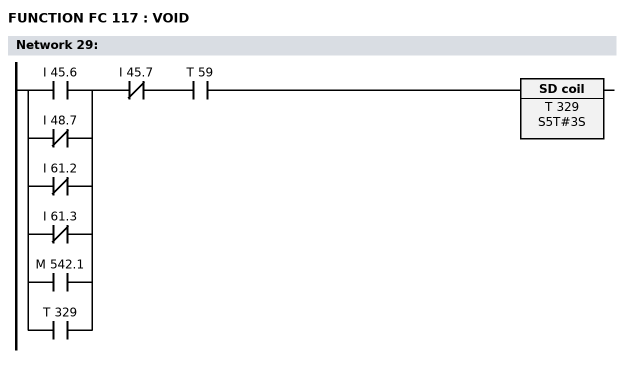

      A(    ;
      O     I     45.6;
      ON    I     48.7;
      ON    I     61.2;
      ON    I     61.3;
      O     M    542.1;
      O     T    329;
      )     ;
      AN    I     45.7;
      A     T     59;
      L     S5T#3S;
      SD    T    329;
NETWORK
TITLE =

      AN    OV;
      =     L      0.0;
      A     L      0.0;
      A     T    329;
      A     M      0.5;
      =     Q     53.6;
      A     L      0.0;
      AN    T    329;
      A(    ;
      O     T    309;
      O     T     69;
      )     ;
      =     Q     53.7;
      A     L      0.0;
      A     I     48.7;
      A     I     61.2;
      A     I     61.3;
      =     L      0.1;
      A     L      0.1;
      A     DB49.DBX    9.2;
      AN    DB49.DBX    9.3;
      =     L      0.2;
      A     L      0.2;
      BLD   102;
      L     S5T#3S;
      SD    T    309;
      A     L      0.2;
      A     T    309;
      =     DB49.DBX    9.4;
      A     L      0.1;
      A     DB49.DBX    9.3;
      AN    DB49.DBX    9.2;
      =     L      0.2;
      A     L      0.2;
      BLD   102;
      L     S5T#3S;
      SD    T     69;
      A     L      0.2;
      A     T     69;
      =     DB49.DBX    9.5;
NETWORK
TITLE =
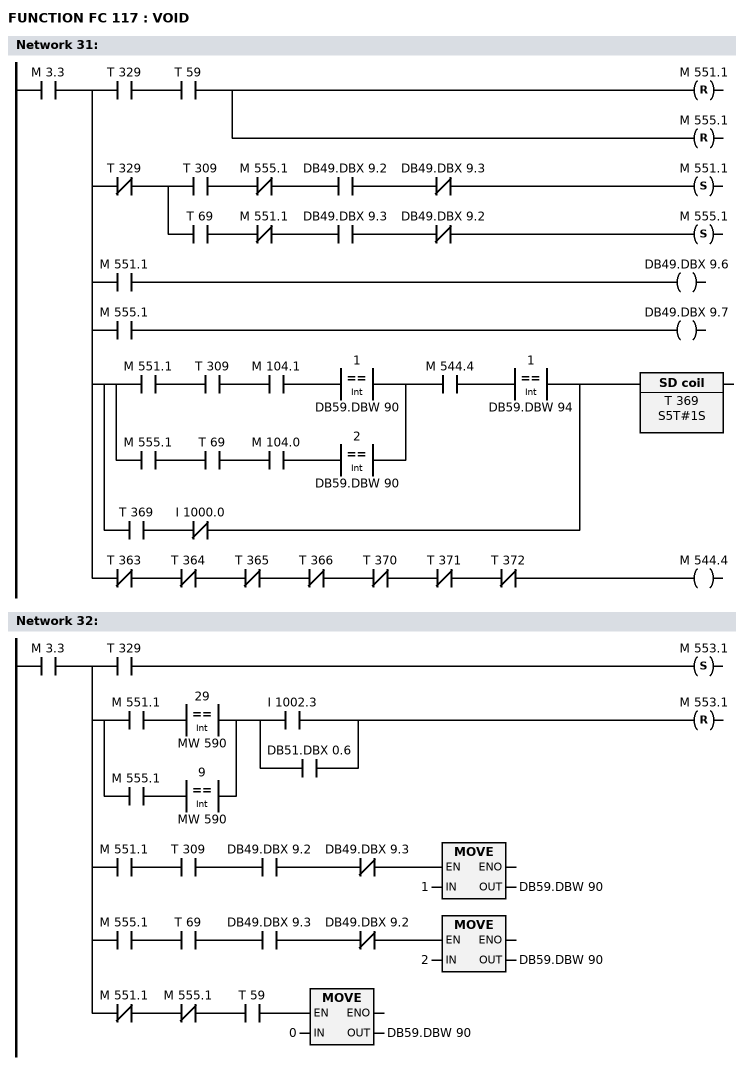

      A     M      3.3;
      =     L      0.0;
      A     L      0.0;
      A     T    329;
      A     T     59;
      R     M    551.1;
      R     M    555.1;
      A     L      0.0;
      AN    T    329;
      =     L      0.1;
      A     L      0.1;
      A     T    309;
      AN    M    555.1;
      A     DB49.DBX    9.2;
      AN    DB49.DBX    9.3;
      S     M    551.1;
      A     L      0.1;
      A     T     69;
      AN    M    551.1;
      A     DB49.DBX    9.3;
      AN    DB49.DBX    9.2;
      S     M    555.1;
      A     L      0.0;
      A     M    551.1;
      =     DB49.DBX    9.6;
      A     L      0.0;
      A     M    555.1;
      =     DB49.DBX    9.7;
      A     L      0.0;
      A(    ;
      A(    ;
      A     M    551.1;
      A     T    309;
      A     M    104.1;
      A(    ;
      L     1;
      L     DB59.DBW   90;
      ==I   ;
      )     ;
      O     ;
      A     M    555.1;
      A     T     69;
      A     M    104.0;
      A(    ;
      L     2;
      L     DB59.DBW   90;
      ==I   ;
      )     ;
      )     ;
      A     M    544.4;
      A(    ;
      L     1;
      L     DB59.DBW   94;
      ==I   ;
      )     ;
      O     ;
      A     T    369;
      AN    I   1000.0;
      )     ;
      L     S5T#1S;
      SD    T    369;
      A     L      0.0;
      AN    T    363;
      AN    T    364;
      AN    T    365;
      AN    T    366;
      AN    T    370;
      AN    T    371;
      AN    T    372;
      =     M    544.4;
NETWORK
TITLE =

      A     M      3.3;
      =     L      0.0;
      A     L      0.0;
      A     T    329;
      S     M    553.1;
      A     L      0.0;
      A(    ;
      A     M    551.1;
      A(    ;
      L     29;
      L     MW   590;
      ==I   ;
      )     ;
      O     ;
      A     M    555.1;
      A(    ;
      L     9;
      L     MW   590;
      ==I   ;
      )     ;
      )     ;
      A(    ;
      O     I   1002.3;
      O     DB51.DBX    0.6;
      )     ;
      R     M    553.1;
      A     L      0.0;
      A     M    551.1;
      A     T    309;
      A     DB49.DBX    9.2;
      AN    DB49.DBX    9.3;
      JNB   _00d;
      L     1;
      T     DB59.DBW   90;
_00d: NOP   0;
      A     L      0.0;
      A     M    555.1;
      A     T     69;
      A     DB49.DBX    9.3;
      AN    DB49.DBX    9.2;
      JNB   _00e;
      L     2;
      T     DB59.DBW   90;
_00e: NOP   0;
      A     L      0.0;
      AN    M    551.1;
      AN    M    555.1;
      A     T     59;
      JNB   _00f;
      L     0;
      T     DB59.DBW   90;
_00f: NOP   0;
NETWORK
TITLE =

      AN    OV;
      =     L      0.0;
      A     L      0.0;
      A(    ;
      A     T    330;
      A     DB49.DBX    2.1;
      A     DB49.DBX   10.0;
      O     ;
      A     M    580.0;
      A     M    580.1;
      O     ;
      AN    M    580.0;
      AN    M    580.1;
      )     ;
      S     M    580.0;
      R     M    580.1;
      A     L      0.0;
      A     T    330;
      A     DB49.DBX    2.1;
      A     DB49.DBX   10.1;
      S     M    580.1;
      R     M    580.0;
      A     L      0.0;
      A     M    580.0;
      =     DB49.DBX   10.2;
      A     L      0.0;
      A     M    580.1;
      =     DB49.DBX   10.3;
NETWORK
TITLE =

      AN    OV;
      =     L      0.0;
      A     L      0.0;
      A(    ;
      A     I     62.0;
      AN    I     62.1;
      O     ;
      AN    I     62.0;
      A     I     62.1;
      O     ;
      AN    I     62.0;
      AN    I     62.1;
      A     I     49.3;
      )     ;
      =     L      0.1;
      A     L      0.1;
      A     T    350;
      =     DB49.DBX    0.5;
      A     L      0.1;
      BLD   102;
      L     S5T#2S;
      SD    T    350;
      A     L      0.0;
      A(    ;
      A     DB49.DBX   10.2;
      A     I     61.1;
      O     ;
      A     DB49.DBX   10.3;
      AN    I     61.1;
      )     ;
      A     I     62.0;
      A     I     62.1;
      A     I     49.3;
      AN    T    330;
      =     L      0.1;
      A     L      0.1;
      A     T    420;
      =     DB49.DBX    1.5;
      A     L      0.1;
      BLD   102;
      L     S5T#3S;
      SD    T    420;
NETWORK
TITLE =
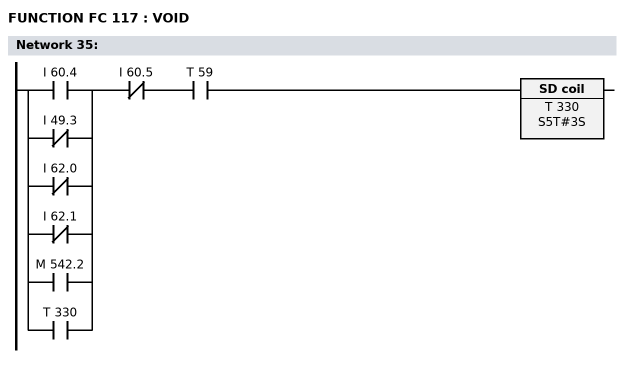

      A(    ;
      O     I     60.4;
      ON    I     49.3;
      ON    I     62.0;
      ON    I     62.1;
      O     M    542.2;
      O     T    330;
      )     ;
      AN    I     60.5;
      A     T     59;
      L     S5T#3S;
      SD    T    330;
NETWORK
TITLE =

      AN    OV;
      =     L      0.0;
      A     L      0.0;
      A     T    330;
      A     M      0.5;
      =     Q     56.4;
      A     L      0.0;
      AN    T    330;
      A(    ;
      O     T    310;
      O     T     70;
      )     ;
      =     Q     56.5;
      A     L      0.0;
      A     I     49.3;
      A     I     62.0;
      A     I     62.1;
      =     L      0.1;
      A     L      0.1;
      A     DB49.DBX   10.2;
      AN    DB49.DBX   10.3;
      =     L      0.2;
      A     L      0.2;
      BLD   102;
      L     S5T#3S;
      SD    T    310;
      A     L      0.2;
      A     T    310;
      =     DB49.DBX   10.4;
      A     L      0.1;
      A     DB49.DBX   10.3;
      AN    DB49.DBX   10.2;
      =     L      0.2;
      A     L      0.2;
      BLD   102;
      L     S5T#3S;
      SD    T     70;
      A     L      0.2;
      A     T     70;
      =     DB49.DBX   10.5;
NETWORK
TITLE =
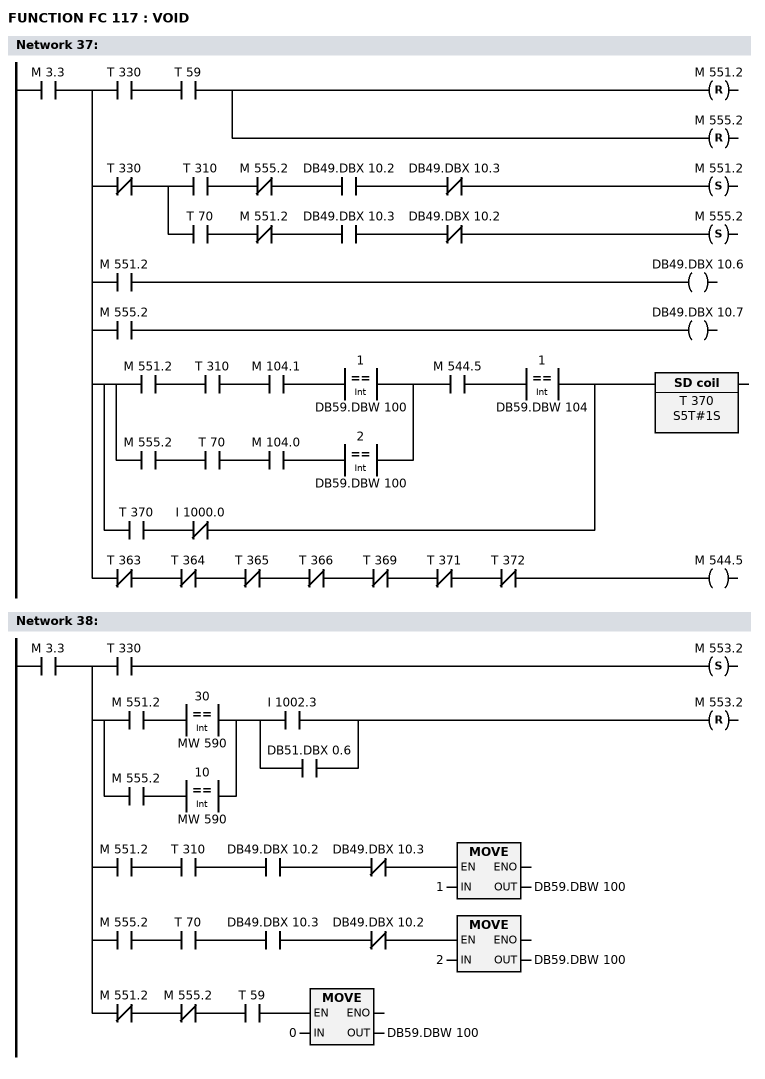

      A     M      3.3;
      =     L      0.0;
      A     L      0.0;
      A     T    330;
      A     T     59;
      R     M    551.2;
      R     M    555.2;
      A     L      0.0;
      AN    T    330;
      =     L      0.1;
      A     L      0.1;
      A     T    310;
      AN    M    555.2;
      A     DB49.DBX   10.2;
      AN    DB49.DBX   10.3;
      S     M    551.2;
      A     L      0.1;
      A     T     70;
      AN    M    551.2;
      A     DB49.DBX   10.3;
      AN    DB49.DBX   10.2;
      S     M    555.2;
      A     L      0.0;
      A     M    551.2;
      =     DB49.DBX   10.6;
      A     L      0.0;
      A     M    555.2;
      =     DB49.DBX   10.7;
      A     L      0.0;
      A(    ;
      A(    ;
      A     M    551.2;
      A     T    310;
      A     M    104.1;
      A(    ;
      L     1;
      L     DB59.DBW  100;
      ==I   ;
      )     ;
      O     ;
      A     M    555.2;
      A     T     70;
      A     M    104.0;
      A(    ;
      L     2;
      L     DB59.DBW  100;
      ==I   ;
      )     ;
      )     ;
      A     M    544.5;
      A(    ;
      L     1;
      L     DB59.DBW  104;
      ==I   ;
      )     ;
      O     ;
      A     T    370;
      AN    I   1000.0;
      )     ;
      L     S5T#1S;
      SD    T    370;
      A     L      0.0;
      AN    T    363;
      AN    T    364;
      AN    T    365;
      AN    T    366;
      AN    T    369;
      AN    T    371;
      AN    T    372;
      =     M    544.5;
NETWORK
TITLE =

      A     M      3.3;
      =     L      0.0;
      A     L      0.0;
      A     T    330;
      S     M    553.2;
      A     L      0.0;
      A(    ;
      A     M    551.2;
      A(    ;
      L     30;
      L     MW   590;
      ==I   ;
      )     ;
      O     ;
      A     M    555.2;
      A(    ;
      L     10;
      L     MW   590;
      ==I   ;
      )     ;
      )     ;
      A(    ;
      O     I   1002.3;
      O     DB51.DBX    0.6;
      )     ;
      R     M    553.2;
      A     L      0.0;
      A     M    551.2;
      A     T    310;
      A     DB49.DBX   10.2;
      AN    DB49.DBX   10.3;
      JNB   _010;
      L     1;
      T     DB59.DBW  100;
_010: NOP   0;
      A     L      0.0;
      A     M    555.2;
      A     T     70;
      A     DB49.DBX   10.3;
      AN    DB49.DBX   10.2;
      JNB   _011;
      L     2;
      T     DB59.DBW  100;
_011: NOP   0;
      A     L      0.0;
      AN    M    551.2;
      AN    M    555.2;
      A     T     59;
      JNB   _012;
      L     0;
      T     DB59.DBW  100;
_012: NOP   0;
NETWORK
TITLE =

      AN    OV;
      =     L      0.0;
      A     L      0.0;
      A(    ;
      A     T    331;
      A     DB49.DBX    2.1;
      A     DB49.DBX   11.0;
      O     ;
      A     M    581.0;
      A     M    581.1;
      O     ;
      AN    M    581.0;
      AN    M    581.1;
      )     ;
      S     M    581.0;
      R     M    581.1;
      A     L      0.0;
      A     T    331;
      A     DB49.DBX    2.1;
      A     DB49.DBX   11.1;
      S     M    581.1;
      R     M    581.0;
      A     L      0.0;
      A     M    581.0;
      =     DB49.DBX   11.2;
      A     L      0.0;
      A     M    581.1;
      =     DB49.DBX   11.3;
NETWORK
TITLE =

      AN    OV;
      =     L      0.0;
      A     L      0.0;
      A(    ;
      A     I     61.4;
      AN    I     61.5;
      O     ;
      AN    I     61.4;
      A     I     61.5;
      O     ;
      AN    I     61.4;
      AN    I     61.5;
      A     I     49.0;
      )     ;
      =     L      0.1;
      A     L      0.1;
      A     T    351;
      =     DB49.DBX    0.6;
      A     L      0.1;
      BLD   102;
      L     S5T#2S;
      SD    T    351;
      A     L      0.0;
      A(    ;
      A     DB49.DBX   11.2;
      A     I     61.6;
      O     ;
      A     DB49.DBX   11.3;
      AN    I     61.6;
      )     ;
      A     I     61.4;
      A     I     61.5;
      A     I     49.0;
      AN    T    331;
      =     L      0.1;
      A     L      0.1;
      A     T    421;
      =     DB49.DBX    1.6;
      A     L      0.1;
      BLD   102;
      L     S5T#3S;
      SD    T    421;
NETWORK
TITLE =
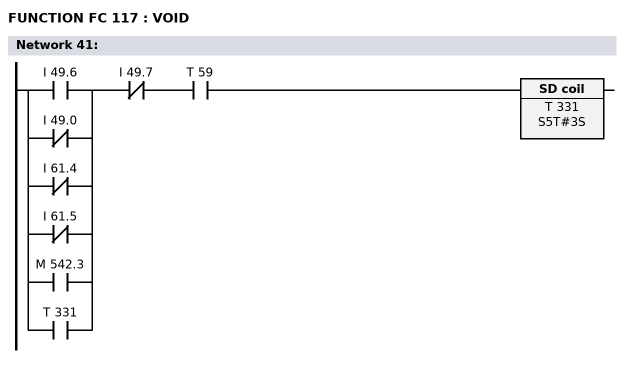

      A(    ;
      O     I     49.6;
      ON    I     49.0;
      ON    I     61.4;
      ON    I     61.5;
      O     M    542.3;
      O     T    331;
      )     ;
      AN    I     49.7;
      A     T     59;
      L     S5T#3S;
      SD    T    331;
NETWORK
TITLE =

      AN    OV;
      =     L      0.0;
      A     L      0.0;
      A     T    331;
      A     M      0.5;
      =     Q     56.0;
      A     L      0.0;
      AN    T    331;
      A(    ;
      O     T    311;
      O     T     71;
      )     ;
      =     Q     56.1;
      A     L      0.0;
      A     I     49.0;
      A     I     61.4;
      A     I     61.5;
      =     L      0.1;
      A     L      0.1;
      A     DB49.DBX   11.2;
      AN    DB49.DBX   11.3;
      =     L      0.2;
      A     L      0.2;
      BLD   102;
      L     S5T#3S;
      SD    T    311;
      A     L      0.2;
      A     T    311;
      =     DB49.DBX   11.4;
      A     L      0.1;
      A     DB49.DBX   11.3;
      AN    DB49.DBX   11.2;
      =     L      0.2;
      A     L      0.2;
      BLD   102;
      L     S5T#3S;
      SD    T     71;
      A     L      0.2;
      A     T     71;
      =     DB49.DBX   11.5;
NETWORK
TITLE =
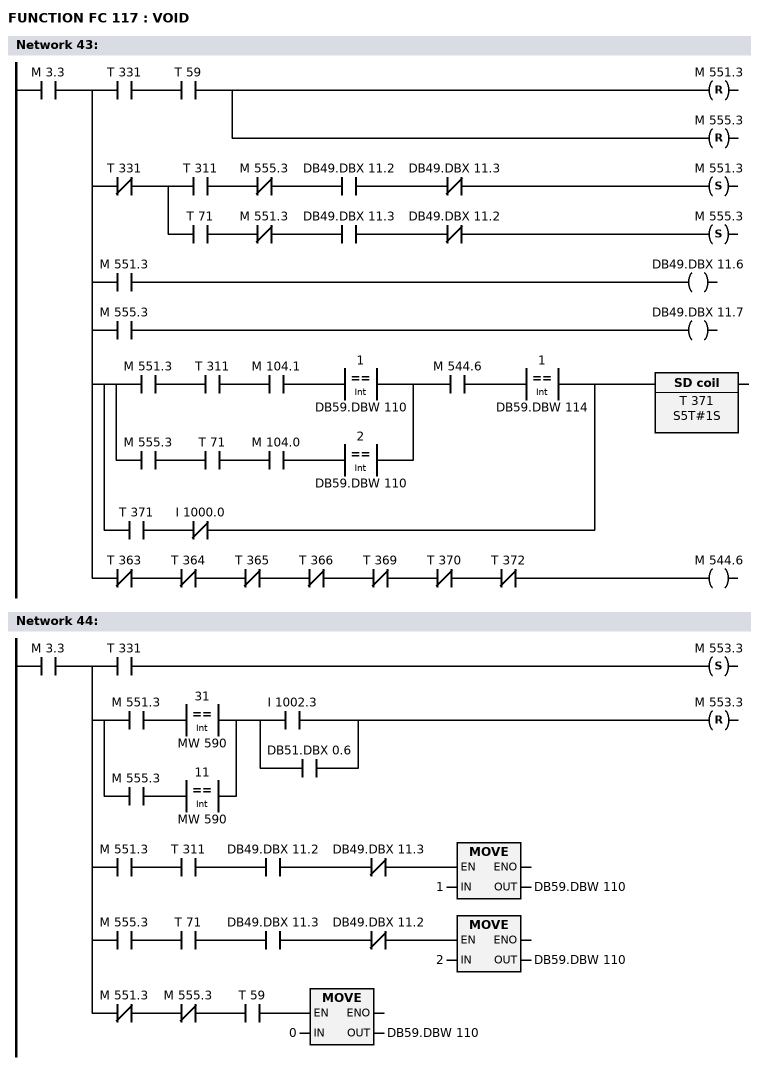

      A     M      3.3;
      =     L      0.0;
      A     L      0.0;
      A     T    331;
      A     T     59;
      R     M    551.3;
      R     M    555.3;
      A     L      0.0;
      AN    T    331;
      =     L      0.1;
      A     L      0.1;
      A     T    311;
      AN    M    555.3;
      A     DB49.DBX   11.2;
      AN    DB49.DBX   11.3;
      S     M    551.3;
      A     L      0.1;
      A     T     71;
      AN    M    551.3;
      A     DB49.DBX   11.3;
      AN    DB49.DBX   11.2;
      S     M    555.3;
      A     L      0.0;
      A     M    551.3;
      =     DB49.DBX   11.6;
      A     L      0.0;
      A     M    555.3;
      =     DB49.DBX   11.7;
      A     L      0.0;
      A(    ;
      A(    ;
      A     M    551.3;
      A     T    311;
      A     M    104.1;
      A(    ;
      L     1;
      L     DB59.DBW  110;
      ==I   ;
      )     ;
      O     ;
      A     M    555.3;
      A     T     71;
      A     M    104.0;
      A(    ;
      L     2;
      L     DB59.DBW  110;
      ==I   ;
      )     ;
      )     ;
      A     M    544.6;
      A(    ;
      L     1;
      L     DB59.DBW  114;
      ==I   ;
      )     ;
      O     ;
      A     T    371;
      AN    I   1000.0;
      )     ;
      L     S5T#1S;
      SD    T    371;
      A     L      0.0;
      AN    T    363;
      AN    T    364;
      AN    T    365;
      AN    T    366;
      AN    T    369;
      AN    T    370;
      AN    T    372;
      =     M    544.6;
NETWORK
TITLE =

      A     M      3.3;
      =     L      0.0;
      A     L      0.0;
      A     T    331;
      S     M    553.3;
      A     L      0.0;
      A(    ;
      A     M    551.3;
      A(    ;
      L     31;
      L     MW   590;
      ==I   ;
      )     ;
      O     ;
      A     M    555.3;
      A(    ;
      L     11;
      L     MW   590;
      ==I   ;
      )     ;
      )     ;
      A(    ;
      O     I   1002.3;
      O     DB51.DBX    0.6;
      )     ;
      R     M    553.3;
      A     L      0.0;
      A     M    551.3;
      A     T    311;
      A     DB49.DBX   11.2;
      AN    DB49.DBX   11.3;
      JNB   _013;
      L     1;
      T     DB59.DBW  110;
_013: NOP   0;
      A     L      0.0;
      A     M    555.3;
      A     T     71;
      A     DB49.DBX   11.3;
      AN    DB49.DBX   11.2;
      JNB   _014;
      L     2;
      T     DB59.DBW  110;
_014: NOP   0;
      A     L      0.0;
      AN    M    551.3;
      AN    M    555.3;
      A     T     59;
      JNB   _015;
      L     0;
      T     DB59.DBW  110;
_015: NOP   0;
NETWORK
TITLE =

      AN    OV;
      =     L      0.0;
      A     L      0.0;
      A(    ;
      A     T    332;
      A     DB49.DBX    2.1;
      A     DB49.DBX   12.0;
      O     ;
      A     M    582.0;
      A     M    582.1;
      O     ;
      AN    M    582.0;
      AN    M    582.1;
      )     ;
      S     M    582.0;
      R     M    582.1;
      A     L      0.0;
      A     T    332;
      A     DB49.DBX    2.1;
      A     DB49.DBX   12.1;
      S     M    582.1;
      R     M    582.0;
      A     L      0.0;
      A     M    582.0;
      =     DB49.DBX   12.2;
      A     L      0.0;
      A     M    582.1;
      =     DB49.DBX   12.3;
NETWORK
TITLE =

      AN    OV;
      =     L      0.0;
      A     L      0.0;
      A(    ;
      A     I     62.2;
      AN    I     62.3;
      O     ;
      AN    I     62.2;
      A     I     62.3;
      O     ;
      AN    I     62.2;
      AN    I     62.3;
      A     I     49.4;
      )     ;
      =     L      0.1;
      A     L      0.1;
      A     T    352;
      =     DB49.DBX    0.7;
      A     L      0.1;
      BLD   102;
      L     S5T#2S;
      SD    T    352;
      A     L      0.0;
      A(    ;
      A     DB49.DBX   12.2;
      A     I     61.7;
      O     ;
      A     DB49.DBX   12.3;
      AN    I     61.7;
      )     ;
      A     I     62.2;
      A     I     62.3;
      A     I     49.4;
      AN    T    332;
      =     L      0.1;
      A     L      0.1;
      A     T    422;
      =     DB49.DBX    1.7;
      A     L      0.1;
      BLD   102;
      L     S5T#3S;
      SD    T    422;
NETWORK
TITLE =
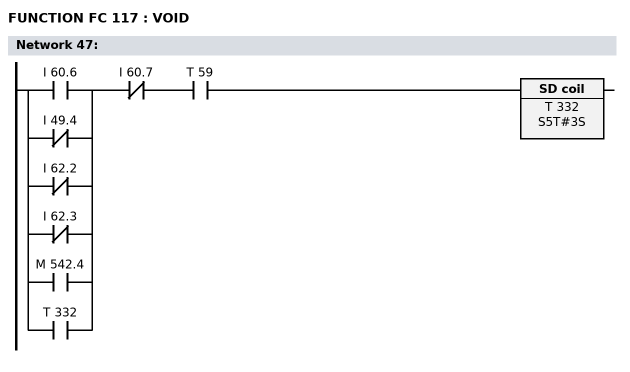

      A(    ;
      O     I     60.6;
      ON    I     49.4;
      ON    I     62.2;
      ON    I     62.3;
      O     M    542.4;
      O     T    332;
      )     ;
      AN    I     60.7;
      A     T     59;
      L     S5T#3S;
      SD    T    332;
NETWORK
TITLE =

      AN    OV;
      =     L      0.0;
      A     L      0.0;
      A     T    332;
      A     M      0.5;
      =     Q     56.6;
      A     L      0.0;
      AN    T    332;
      A(    ;
      O     T    312;
      O     T     72;
      )     ;
      =     Q     56.7;
      A     L      0.0;
      A     I     49.4;
      A     I     62.2;
      A     I     62.3;
      =     L      0.1;
      A     L      0.1;
      A     DB49.DBX   12.2;
      AN    DB49.DBX   12.3;
      =     L      0.2;
      A     L      0.2;
      BLD   102;
      L     S5T#3S;
      SD    T    312;
      A     L      0.2;
      A     T    312;
      =     DB49.DBX   12.4;
      A     L      0.1;
      A     DB49.DBX   12.3;
      AN    DB49.DBX   12.2;
      =     L      0.2;
      A     L      0.2;
      BLD   102;
      L     S5T#3S;
      SD    T     72;
      A     L      0.2;
      A     T     72;
      =     DB49.DBX   12.5;
NETWORK
TITLE =
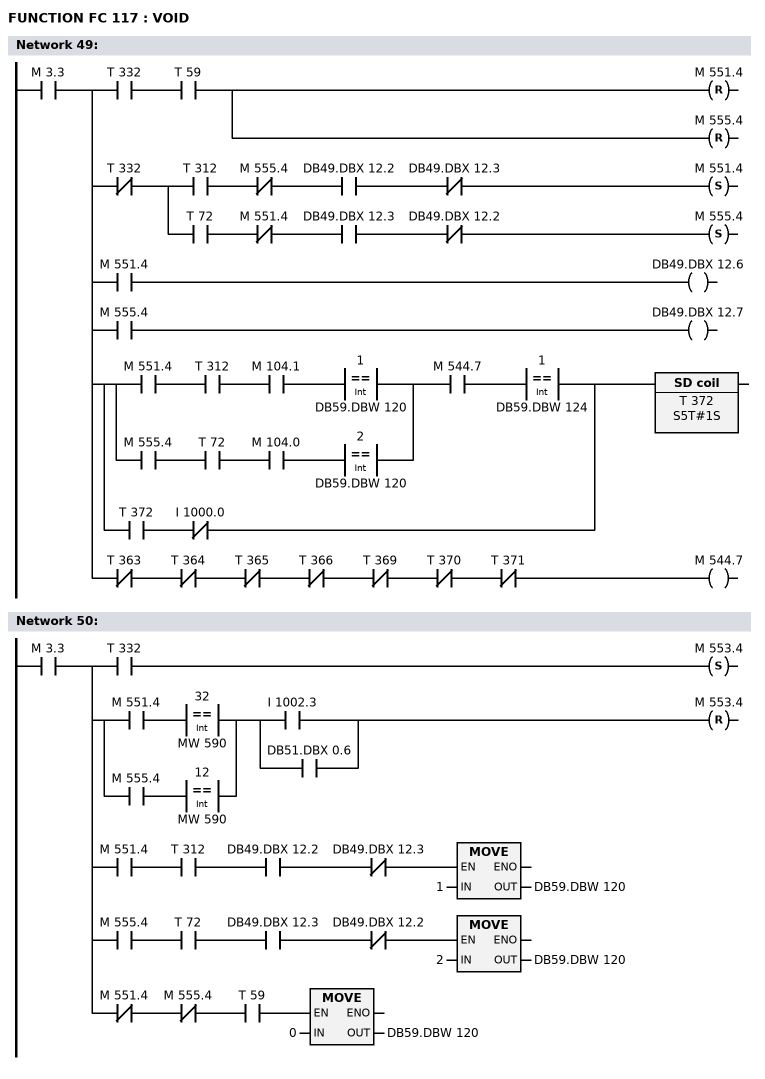

      A     M      3.3;
      =     L      0.0;
      A     L      0.0;
      A     T    332;
      A     T     59;
      R     M    551.4;
      R     M    555.4;
      A     L      0.0;
      AN    T    332;
      =     L      0.1;
      A     L      0.1;
      A     T    312;
      AN    M    555.4;
      A     DB49.DBX   12.2;
      AN    DB49.DBX   12.3;
      S     M    551.4;
      A     L      0.1;
      A     T     72;
      AN    M    551.4;
      A     DB49.DBX   12.3;
      AN    DB49.DBX   12.2;
      S     M    555.4;
      A     L      0.0;
      A     M    551.4;
      =     DB49.DBX   12.6;
      A     L      0.0;
      A     M    555.4;
      =     DB49.DBX   12.7;
      A     L      0.0;
      A(    ;
      A(    ;
      A     M    551.4;
      A     T    312;
      A     M    104.1;
      A(    ;
      L     1;
      L     DB59.DBW  120;
      ==I   ;
      )     ;
      O     ;
      A     M    555.4;
      A     T     72;
      A     M    104.0;
      A(    ;
      L     2;
      L     DB59.DBW  120;
      ==I   ;
      )     ;
      )     ;
      A     M    544.7;
      A(    ;
      L     1;
      L     DB59.DBW  124;
      ==I   ;
      )     ;
      O     ;
      A     T    372;
      AN    I   1000.0;
      )     ;
      L     S5T#1S;
      SD    T    372;
      A     L      0.0;
      AN    T    363;
      AN    T    364;
      AN    T    365;
      AN    T    366;
      AN    T    369;
      AN    T    370;
      AN    T    371;
      =     M    544.7;
NETWORK
TITLE =

      A     M      3.3;
      =     L      0.0;
      A     L      0.0;
      A     T    332;
      S     M    553.4;
      A     L      0.0;
      A(    ;
      A     M    551.4;
      A(    ;
      L     32;
      L     MW   590;
      ==I   ;
      )     ;
      O     ;
      A     M    555.4;
      A(    ;
      L     12;
      L     MW   590;
      ==I   ;
      )     ;
      )     ;
      A(    ;
      O     I   1002.3;
      O     DB51.DBX    0.6;
      )     ;
      R     M    553.4;
      A     L      0.0;
      A     M    551.4;
      A     T    312;
      A     DB49.DBX   12.2;
      AN    DB49.DBX   12.3;
      JNB   _016;
      L     1;
      T     DB59.DBW  120;
_016: NOP   0;
      A     L      0.0;
      A     M    555.4;
      A     T     72;
      A     DB49.DBX   12.3;
      AN    DB49.DBX   12.2;
      JNB   _017;
      L     2;
      T     DB59.DBW  120;
_017: NOP   0;
      A     L      0.0;
      AN    M    551.4;
      AN    M    555.4;
      A     T     59;
      JNB   _018;
      L     0;
      T     DB59.DBW  120;
_018: NOP   0;
NETWORK
TITLE =

      AN    OV;
      =     L      0.0;
      A     L      0.0;
      A     I     45.1;
      L     S5T#3S;
      SD    T    158;
      A     L      0.0;
      A     I     44.3;
      L     S5T#3S;
      SD    T    159;
      A     L      0.0;
      A     I     45.3;
      L     S5T#3S;
      SD    T    160;
      A     L      0.0;
      A     I     44.5;
      L     S5T#3S;
      SD    T    161;
      A     L      0.0;
      A     I     45.7;
      L     S5T#3S;
      SD    T    164;
      A     L      0.0;
      A     I     60.5;
      L     S5T#3S;
      SD    T    165;
      A     L      0.0;
      A     I     49.7;
      L     S5T#3S;
      SD    T    166;
      A     L      0.0;
      A     I     60.7;
      L     S5T#3S;
      SD    T    167;
NETWORK
TITLE =

      AN    OV;
      =     L      0.0;
      A     L      0.0;
      A(    ;
      O(    ;
      L     23;
      L     MW   590;
      ==I   ;
      )     ;
      O(    ;
      L     3;
      L     MW   590;
      ==I   ;
      )     ;
      )     ;
      A     I   1003.6;
      =     M    541.3;
      A     L      0.0;
      A(    ;
      O(    ;
      L     24;
      L     MW   590;
      ==I   ;
      )     ;
      O(    ;
      L     4;
      L     MW   590;
      ==I   ;
      )     ;
      )     ;
      A     I   1003.6;
      =     M    541.4;
      A     L      0.0;
      A(    ;
      O(    ;
      L     25;
      L     MW   590;
      ==I   ;
      )     ;
      O(    ;
      L     5;
      L     MW   590;
      ==I   ;
      )     ;
      )     ;
      A     I   1003.6;
      =     M    541.5;
      A     L      0.0;
      A(    ;
      O(    ;
      L     26;
      L     MW   590;
      ==I   ;
      )     ;
      O(    ;
      L     6;
      L     MW   590;
      ==I   ;
      )     ;
      )     ;
      A     I   1003.6;
      =     M    541.6;
      A     L      0.0;
      A(    ;
      O(    ;
      L     29;
      L     MW   590;
      ==I   ;
      )     ;
      O(    ;
      L     9;
      L     MW   590;
      ==I   ;
      )     ;
      )     ;
      A     I   1003.6;
      =     M    542.1;
      A     L      0.0;
      A(    ;
      O(    ;
      L     30;
      L     MW   590;
      ==I   ;
      )     ;
      O(    ;
      L     10;
      L     MW   590;
      ==I   ;
      )     ;
      )     ;
      A     I   1003.6;
      =     M    542.2;
      A     L      0.0;
      A(    ;
      O(    ;
      L     31;
      L     MW   590;
      ==I   ;
      )     ;
      O(    ;
      L     11;
      L     MW   590;
      ==I   ;
      )     ;
      )     ;
      A     I   1003.6;
      =     M    542.3;
      A     L      0.0;
      A(    ;
      O(    ;
      L     32;
      L     MW   590;
      ==I   ;
      )     ;
      O(    ;
      L     12;
      L     MW   590;
      ==I   ;
      )     ;
      )     ;
      A     I   1003.6;
      =     M    542.4;
NETWORK
TITLE =

      A     M      3.3;
      =     L      0.0;
      BLD   103;
      CALL FB   515 , DB   200 (
           STN_V_ACTIVE             := L      0.0,
           PLT_Amount               := 12,
           PLT1_Code                := 0,
           PLT2_Code                := 0,
           PLT3_Code                := DB59.DBW   30,
           PLT4_Code                := DB59.DBW   40,
           PLT5_Code                := DB59.DBW   50,
           PLT6_Code                := DB59.DBW   60,
           PLT9_Code                := DB59.DBW   90,
           PLT10_Code               := DB59.DBW  100,
           PLT11_Code               := DB59.DBW  110,
           PLT12_Code               := DB59.DBW  120,
           PLT13_Code               := 0,
           PLT14_Code               := 0,
           PLT15_Code               := 0,
           PLT16_Code               := 0,
           PLT17_Code               := 0,
           PLT18_Code               := 0,
           PLT19_Code               := 0,
           PLT20_Code               := 0,
           PLT3_Priority            := DB59.DBW   34,
           PLT4_Priority            := DB59.DBW   44,
           PLT5_Priority            := DB59.DBW   54,
           PLT6_Priority            := DB59.DBW   64,
           PLT9_Priority            := DB59.DBW   94,
           PLT10_Priority           := DB59.DBW  104,
           PLT11_Priority           := DB59.DBW  114,
           PLT12_Priority           := DB59.DBW  124);

      NOP   0;
END_FUNCTION

FUNCTION FC 118 : VOID
TITLE =
VERSION : 0.1

BEGIN
NETWORK
TITLE =
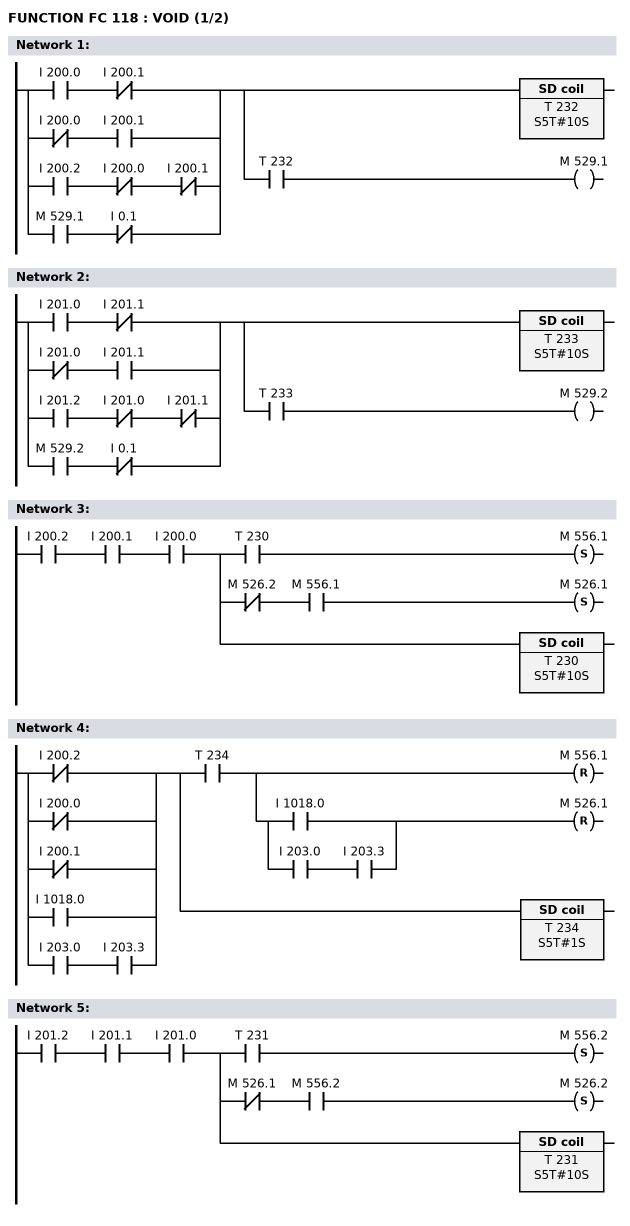

      A     I    200.0;
      AN    I    200.1;
      O     ;
      AN    I    200.0;
      A     I    200.1;
      O     ;
      A     I    200.2;
      AN    I    200.0;
      AN    I    200.1;
      O     ;
      A     M    529.1;
      AN    I      0.1;
      =     L      0.0;
      A     L      0.0;
      BLD   102;
      L     S5T#10S;
      SD    T    232;
      A     L      0.0;
      A     T    232;
      =     M    529.1;
NETWORK
TITLE =

      A     I    201.0;
      AN    I    201.1;
      O     ;
      AN    I    201.0;
      A     I    201.1;
      O     ;
      A     I    201.2;
      AN    I    201.0;
      AN    I    201.1;
      O     ;
      A     M    529.2;
      AN    I      0.1;
      =     L      0.0;
      A     L      0.0;
      BLD   102;
      L     S5T#10S;
      SD    T    233;
      A     L      0.0;
      A     T    233;
      =     M    529.2;
NETWORK
TITLE =

      A     I    200.2;
      A     I    200.1;
      A     I    200.0;
      =     L      0.0;
      A     L      0.0;
      A     T    230;
      S     M    556.1;
      A     L      0.0;
      AN    M    526.2;
      A     M    556.1;
      S     M    526.1;
      A     L      0.0;
      BLD   102;
      L     S5T#10S;
      SD    T    230;
NETWORK
TITLE =

      ON    I    200.2;
      ON    I    200.0;
      ON    I    200.1;
      O     I   1018.0;
      O     ;
      A     I    203.0;
      A     I    203.3;
      =     L      0.0;
      A     L      0.0;
      A     T    234;
      =     L      0.1;
      A     L      0.1;
      BLD   102;
      R     M    556.1;
      A     L      0.1;
      A(    ;
      O     I   1018.0;
      O     ;
      A     I    203.0;
      A     I    203.3;
      )     ;
      R     M    526.1;
      A     L      0.0;
      BLD   102;
      L     S5T#1S;
      SD    T    234;
NETWORK
TITLE =

      A     I    201.2;
      A     I    201.1;
      A     I    201.0;
      =     L      0.0;
      A     L      0.0;
      A     T    231;
      S     M    556.2;
      A     L      0.0;
      AN    M    526.1;
      A     M    556.2;
      S     M    526.2;
      A     L      0.0;
      BLD   102;
      L     S5T#10S;
      SD    T    231;
NETWORK
TITLE =
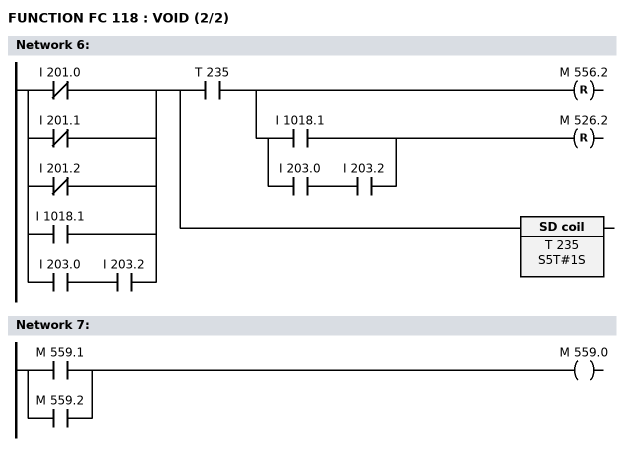

      ON    I    201.0;
      ON    I    201.1;
      ON    I    201.2;
      O     I   1018.1;
      O     ;
      A     I    203.0;
      A     I    203.2;
      =     L      0.0;
      A     L      0.0;
      A     T    235;
      =     L      0.1;
      A     L      0.1;
      BLD   102;
      R     M    556.2;
      A     L      0.1;
      A(    ;
      O     I   1018.1;
      O     ;
      A     I    203.0;
      A     I    203.2;
      )     ;
      R     M    526.2;
      A     L      0.0;
      BLD   102;
      L     S5T#1S;
      SD    T    235;
NETWORK
TITLE =

      O     M    559.1;
      O     M    559.2;
      =     M    559.0;
NETWORK
TITLE =

      AN    OV;
      =     L      0.0;
      A     L      0.0;
      A     M    559.4;
      AN    M    556.1;
      S     M    559.1;
      A     L      0.0;
      A(    ;
      A     M    556.1;
      A     T    230;
      O     ;
      A     I    203.0;
      A     I    203.3;
      O     ;
      AN    I    201.2;
      AN    I    200.0;
      AN    I    200.1;
      O     ;
      AN    I    201.1;
      AN    I    201.0;
      AN    I    200.2;
      )     ;
      R     M    559.1;
NETWORK
TITLE =

      AN    OV;
      =     L      0.0;
      A     L      0.0;
      A     M    559.3;
      AN    M    556.2;
      S     M    559.2;
      A     L      0.0;
      A(    ;
      A     M    556.2;
      A     T    231;
      O     ;
      A     I    203.0;
      A     I    203.2;
      O     ;
      AN    I    200.2;
      AN    I    201.1;
      AN    I    201.0;
      O     ;
      AN    I    200.0;
      AN    I    200.1;
      AN    I    201.2;
      )     ;
      R     M    559.2;
NETWORK
TITLE =
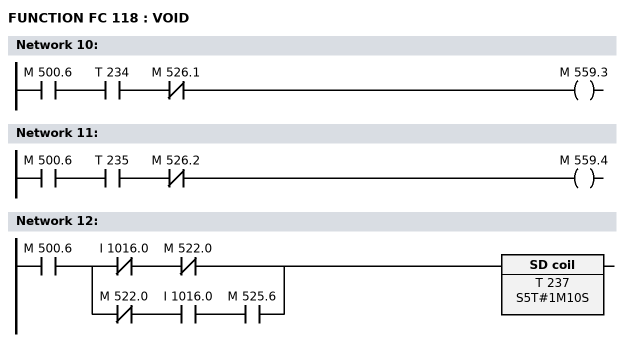

      A     M    500.6;
      A     T    234;
      AN    M    526.1;
      =     M    559.3;
NETWORK
TITLE =

      A     M    500.6;
      A     T    235;
      AN    M    526.2;
      =     M    559.4;
NETWORK
TITLE =

      A     M    500.6;
      A(    ;
      AN    I   1016.0;
      AN    M    522.0;
      O     ;
      AN    M    522.0;
      A     I   1016.0;
      A     M    525.6;
      )     ;
      L     S5T#1M10S;
      SD    T    237;
NETWORK
TITLE =

      AN    OV;
      =     L      0.0;
      A     L      0.0;
      AN    I    203.1;
      A     M      0.5;
      =     Q    205.2;
      A     L      0.0;
      A(    ;
      O     M    526.1;
      O     ;
      A     T    230;
      AN    M    526.1;
      A     M      0.5;
      )     ;
      =     Q    205.0;
      A     L      0.0;
      A(    ;
      O     M    526.2;
      O     ;
      A     T    231;
      AN    M    526.2;
      A     M      0.5;
      )     ;
      =     Q    205.1;
      A     L      0.0;
      A(    ;
      A     T    230;
      A     T    231;
      O     ;
      A(    ;
      ON    T    230;
      ON    T    231;
      )     ;
      A     M      0.5;
      )     ;
      =     Q    205.3;
NETWORK
TITLE =
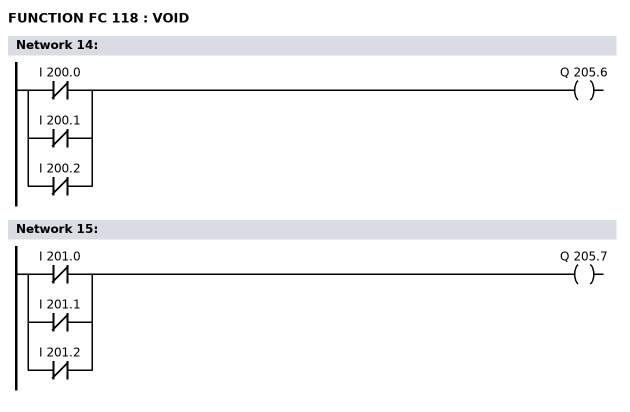

      ON    I    200.0;
      ON    I    200.1;
      ON    I    200.2;
      =     Q    205.6;
NETWORK
TITLE =

      ON    I    201.0;
      ON    I    201.1;
      ON    I    201.2;
      =     Q    205.7;
END_FUNCTION

FUNCTION_BLOCK FB 120
TITLE =
VERSION : 0.1


VAR
  S701_STN_MODE : FB 402;	//S701_STN_MODE
END_VAR
BEGIN
NETWORK
TITLE =
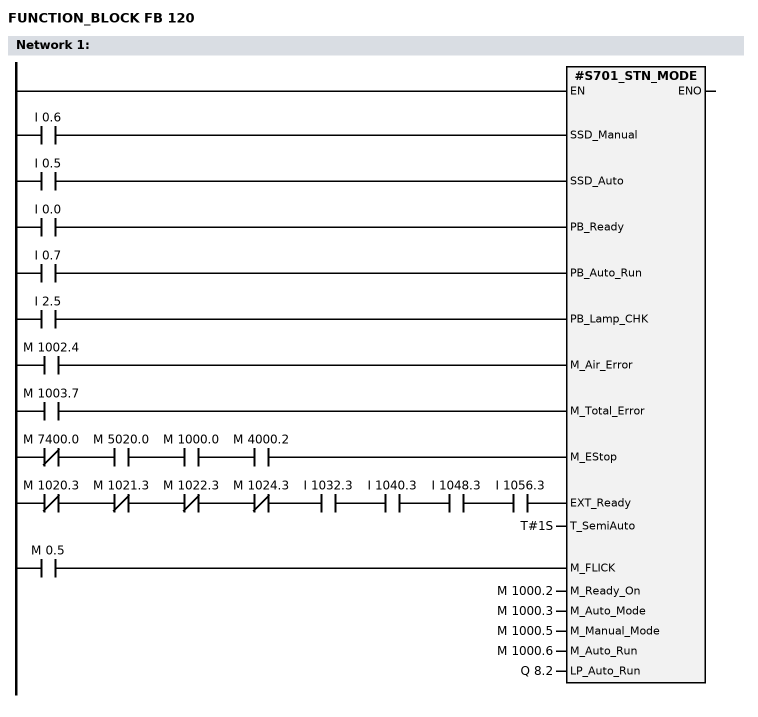

      A     I      0.6;
      =     L      0.0;
      BLD   103;
      A     I      0.5;
      =     L      0.1;
      BLD   103;
      A     I      0.0;
      =     L      0.2;
      BLD   103;
      A     I      0.7;
      =     L      0.3;
      BLD   103;
      A     I      2.5;
      =     L      0.6;
      BLD   103;
      A     M   1002.4;
      =     L      0.7;
      BLD   103;
      A     M   1003.7;
      =     L      1.1;
      BLD   103;
      AN    M   7400.0;
      A     M   5020.0;
      A     M   1000.0;
      A     M   4000.2;
      =     L      1.2;
      BLD   103;
      AN    M   1020.3;
      AN    M   1021.3;
      AN    M   1022.3;
      AN    M   1024.3;
      A     I   1032.3;
      A     I   1040.3;
      A     I   1048.3;
      A     I   1056.3;
      =     L      1.3;
      BLD   103;
      A     M      0.5;
      =     L      1.5;
      BLD   103;
      CALL #S701_STN_MODE (
           SSD_Manual               := L      0.0,
           SSD_Auto                 := L      0.1,
           PB_Ready                 := L      0.2,
           PB_Auto_Run              := L      0.3,
           PB_Lamp_CHK              := L      0.6,
           M_Air_Error              := L      0.7,
           M_Total_Error            := L      1.1,
           M_EStop                  := L      1.2,
           EXT_Ready                := L      1.3,
           T_SemiAuto               := T#1S,
           M_FLICK                  := L      1.5,
           M_Ready_On               := M   1000.2,
           M_Auto_Mode              := M   1000.3,
           M_Manual_Mode            := M   1000.5,
           M_Auto_Run               := M   1000.6,
           LP_Auto_Run              := Q      8.2);
      NOP   0;
END_FUNCTION_BLOCK

DATA_BLOCK DB 120
TITLE =
VERSION : 0.0

 FB 120
BEGIN
   S701_STN_MODE.SSD_Manual := FALSE;
   S701_STN_MODE.SSD_Auto := FALSE;
   S701_STN_MODE.PB_Ready := FALSE;
   S701_STN_MODE.PB_Auto_Run := FALSE;
   S701_STN_MODE.PB_Remote_Ready := FALSE;
   S701_STN_MODE.PB_Remote_Auto_Run := FALSE;
   S701_STN_MODE.PB_Lamp_CHK := FALSE;
   S701_STN_MODE.M_Air_Error := FALSE;
   S701_STN_MODE.M_Water_Error := FALSE;
   S701_STN_MODE.M_Total_Error := FALSE;
   S701_STN_MODE.M_EStop := FALSE;
   S701_STN_MODE.EXT_Ready := FALSE;
   S701_STN_MODE.EXT_Auto := FALSE;
   S701_STN_MODE.T_SemiAuto := T#0MS;
   S701_STN_MODE.M_FLICK := FALSE;
   S701_STN_MODE.M_Ready_On := FALSE;
   S701_STN_MODE.M_Auto_Mode := FALSE;
   S701_STN_MODE.M_SemiAuto_Mode := FALSE;
   S701_STN_MODE.M_Manual_Mode := FALSE;
   S701_STN_MODE.M_Auto_Run := FALSE;
   S701_STN_MODE.LP_Ready_On := FALSE;
   S701_STN_MODE.LP_Auto_Run := FALSE;
   S701_STN_MODE.AUTO_MODE_DELAY.IN := FALSE;
   S701_STN_MODE.AUTO_MODE_DELAY.PT := T#0MS;
   S701_STN_MODE.AUTO_MODE_DELAY.Q := FALSE;
   S701_STN_MODE.AUTO_MODE_DELAY.ET := T#0MS;
   S701_STN_MODE.AUTO_MODE_DELAY.STATE := B#16#0;
   S701_STN_MODE.AUTO_MODE_DELAY.STIME := T#0MS;
   S701_STN_MODE.AUTO_MODE_DELAY.ATIME := T#0MS;
   S701_STN_MODE.SEMI_AUTO_DELAY.IN := FALSE;
   S701_STN_MODE.SEMI_AUTO_DELAY.PT := T#0MS;
   S701_STN_MODE.SEMI_AUTO_DELAY.Q := FALSE;
   S701_STN_MODE.SEMI_AUTO_DELAY.ET := T#0MS;
   S701_STN_MODE.SEMI_AUTO_DELAY.STATE := B#16#0;
   S701_STN_MODE.SEMI_AUTO_DELAY.STIME := T#0MS;
   S701_STN_MODE.SEMI_AUTO_DELAY.ATIME := T#0MS;
   S701_STN_MODE.MANUAL_DELAY.IN := FALSE;
   S701_STN_MODE.MANUAL_DELAY.PT := T#0MS;
   S701_STN_MODE.MANUAL_DELAY.Q := FALSE;
   S701_STN_MODE.MANUAL_DELAY.ET := T#0MS;
   S701_STN_MODE.MANUAL_DELAY.STATE := B#16#0;
   S701_STN_MODE.MANUAL_DELAY.STIME := T#0MS;
   S701_STN_MODE.MANUAL_DELAY.ATIME := T#0MS;
END_DATA_BLOCK

FUNCTION FC 120 : VOID
TITLE =
VERSION : 0.1

BEGIN
NETWORK
TITLE =
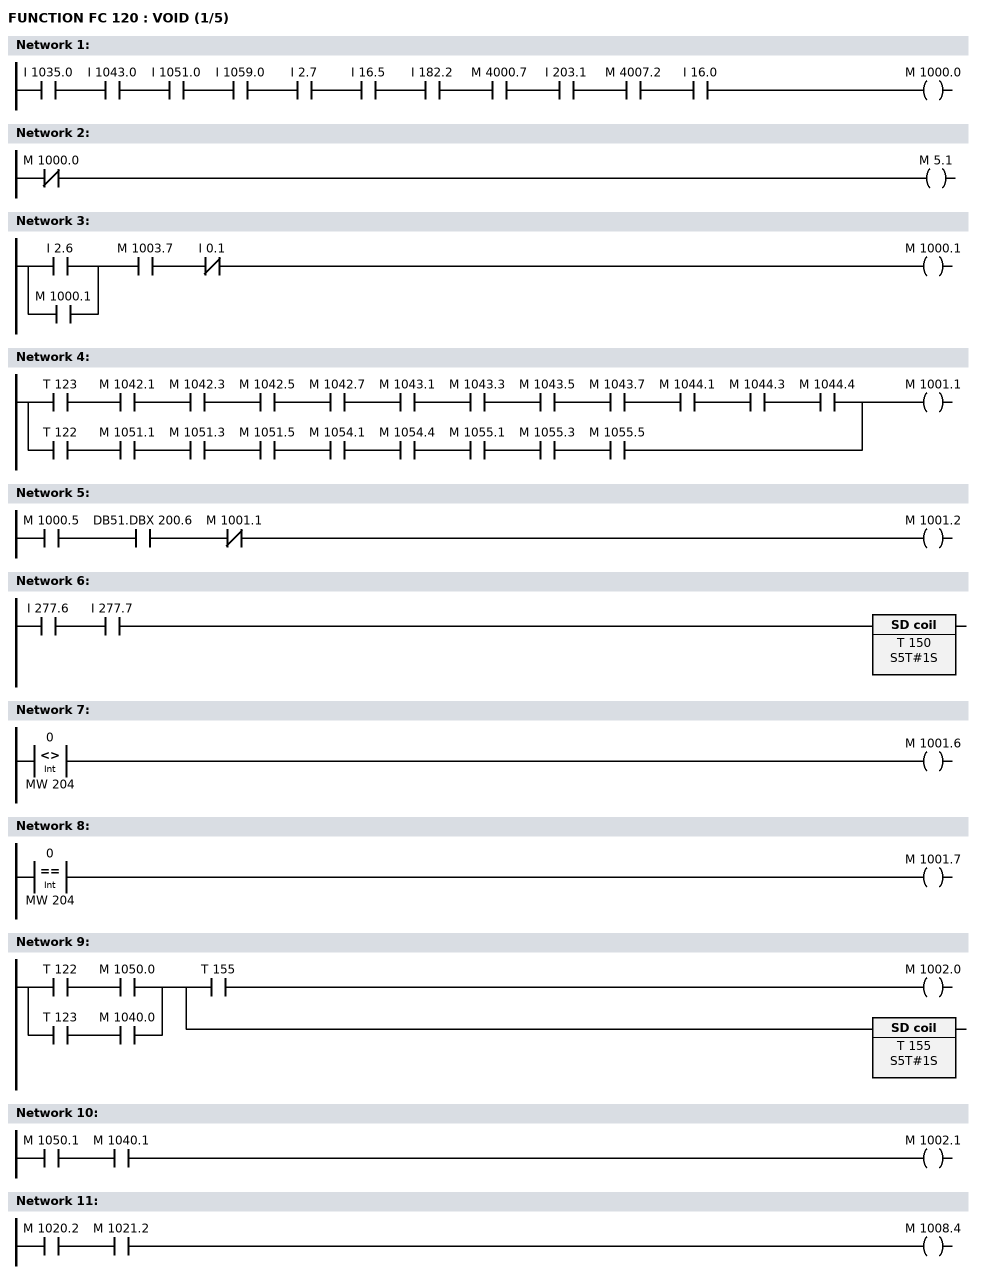

      A     I   1035.0;
      A     I   1043.0;
      A     I   1051.0;
      A     I   1059.0;
      A     I      2.7;
      A     I     16.5;
      A     I    182.2;
      A     M   4000.7;
      A     I    203.1;
      A     M   4007.2;
      A     I     16.0;
      =     M   1000.0;
NETWORK
TITLE =

      AN    M   1000.0;
      =     M      5.1;
NETWORK
TITLE =

      A(    ;
      O     I      2.6;
      O     M   1000.1;
      )     ;
      A     M   1003.7;
      AN    I      0.1;
      =     M   1000.1;
NETWORK
TITLE =

      A     T    123;
      A     M   1042.1;
      A     M   1042.3;
      A     M   1042.5;
      A     M   1042.7;
      A     M   1043.1;
      A     M   1043.3;
      A     M   1043.5;
      A     M   1043.7;
      A     M   1044.1;
      A     M   1044.3;
      A     M   1044.4;
      O     ;
      A     T    122;
      A     M   1051.1;
      A     M   1051.3;
      A     M   1051.5;
      A     M   1054.1;
      A     M   1054.4;
      A     M   1055.1;
      A     M   1055.3;
      A     M   1055.5;
      =     M   1001.1;
NETWORK
TITLE =

      A     M   1000.5;
      A     DB51.DBX  200.6;
      AN    M   1001.1;
      =     M   1001.2;
NETWORK
TITLE =

      A     I    277.6;
      A     I    277.7;
      L     S5T#1S;
      SD    T    150;
NETWORK
TITLE =

      L     0;
      L     MW   204;
      <>I   ;
      =     M   1001.6;
NETWORK
TITLE =

      L     0;
      L     MW   204;
      ==I   ;
      =     M   1001.7;
NETWORK
TITLE =

      A     T    122;
      A     M   1050.0;
      O     ;
      A     T    123;
      A     M   1040.0;
      =     L      0.0;
      A     L      0.0;
      A     T    155;
      =     M   1002.0;
      A     L      0.0;
      BLD   102;
      L     S5T#1S;
      SD    T    155;
NETWORK
TITLE =

      A     M   1050.1;
      A     M   1040.1;
      =     M   1002.1;
NETWORK
TITLE =

      A     M   1020.2;
      A     M   1021.2;
      =     M   1008.4;
NETWORK
TITLE =
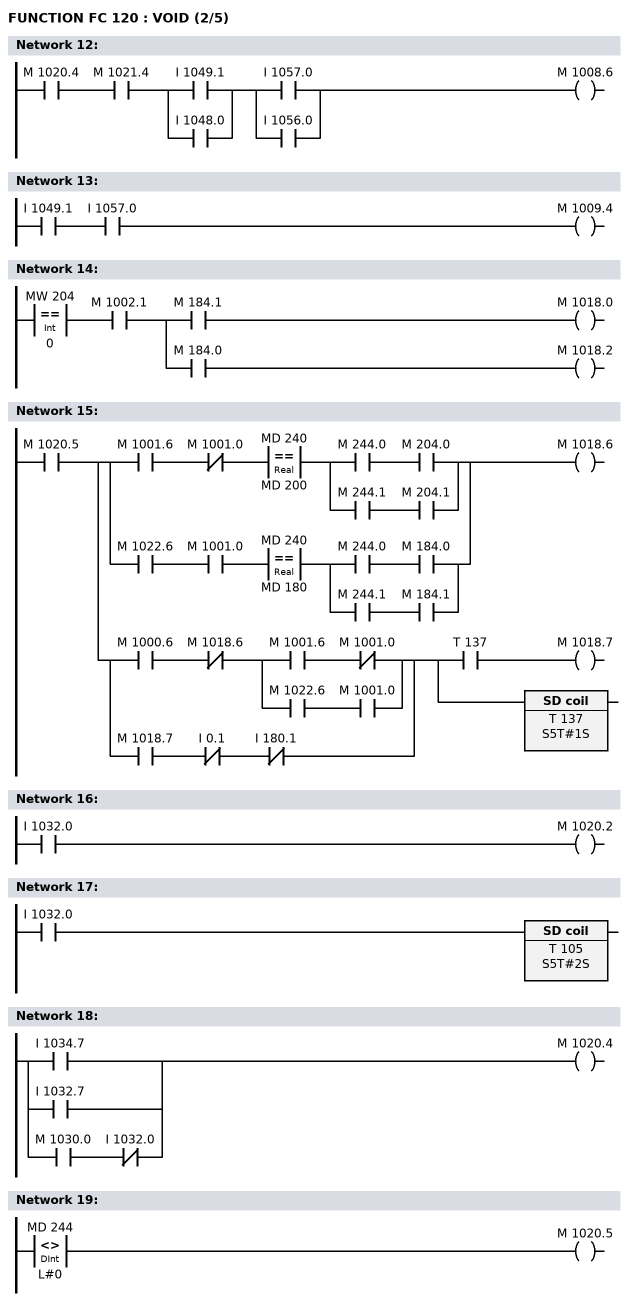

      A     M   1020.4;
      A     M   1021.4;
      A(    ;
      O     I   1049.1;
      O     I   1048.0;
      )     ;
      A(    ;
      O     I   1057.0;
      O     I   1056.0;
      )     ;
      =     M   1008.6;
NETWORK
TITLE =

      A     I   1049.1;
      A     I   1057.0;
      =     M   1009.4;
NETWORK
TITLE =

      A(    ;
      L     MW   204;
      L     0;
      ==I   ;
      )     ;
      A     M   1002.1;
      =     L      0.0;
      A     L      0.0;
      A     M    184.1;
      =     M   1018.0;
      A     L      0.0;
      A     M    184.0;
      =     M   1018.2;
NETWORK
TITLE =

      A     M   1020.5;
      =     L      0.0;
      A     L      0.0;
      A(    ;
      A     M   1001.6;
      AN    M   1001.0;
      A(    ;
      L     MD   240;
      L     MD   200;
      ==R   ;
      )     ;
      A(    ;
      A     M    244.0;
      A     M    204.0;
      O     ;
      A     M    244.1;
      A     M    204.1;
      )     ;
      O     ;
      A     M   1022.6;
      A     M   1001.0;
      A(    ;
      L     MD   240;
      L     MD   180;
      ==R   ;
      )     ;
      A(    ;
      A     M    244.0;
      A     M    184.0;
      O     ;
      A     M    244.1;
      A     M    184.1;
      )     ;
      )     ;
      =     M   1018.6;
      A     L      0.0;
      A(    ;
      A     M   1000.6;
      AN    M   1018.6;
      A(    ;
      A     M   1001.6;
      AN    M   1001.0;
      O     ;
      A     M   1022.6;
      A     M   1001.0;
      )     ;
      O     ;
      A     M   1018.7;
      AN    I      0.1;
      AN    I    180.1;
      )     ;
      =     L      0.1;
      A     L      0.1;
      A     T    137;
      =     M   1018.7;
      A     L      0.1;
      BLD   102;
      L     S5T#1S;
      SD    T    137;
NETWORK
TITLE =

      A     I   1032.0;
      =     M   1020.2;
NETWORK
TITLE =

      A     I   1032.0;
      L     S5T#2S;
      SD    T    105;
NETWORK
TITLE =

      O     I   1034.7;
      O     I   1032.7;
      O     ;
      A     M   1030.0;
      AN    I   1032.0;
      =     M   1020.4;
NETWORK
TITLE =

      L     MD   244;
      L     L#0;
      <>D   ;
      =     M   1020.5;
NETWORK
TITLE =
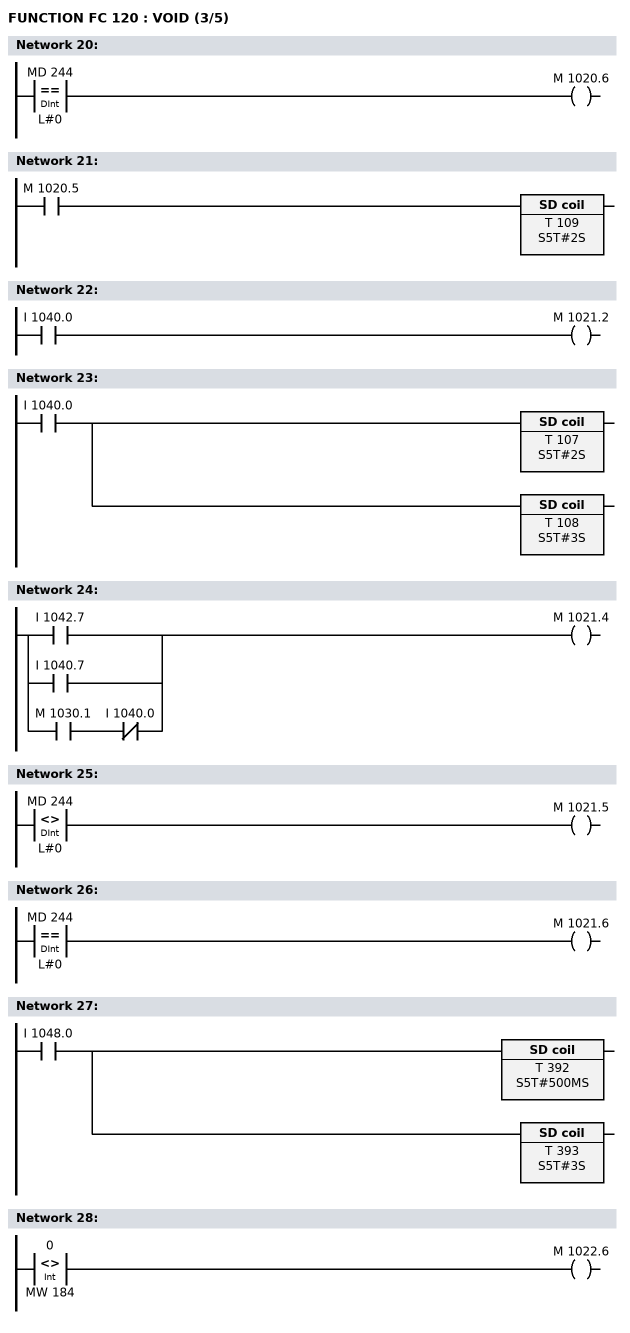

      L     MD   244;
      L     L#0;
      ==D   ;
      =     M   1020.6;
NETWORK
TITLE =

      A     M   1020.5;
      L     S5T#2S;
      SD    T    109;
NETWORK
TITLE =

      A     I   1040.0;
      =     M   1021.2;
NETWORK
TITLE =

      A     I   1040.0;
      L     S5T#2S;
      SD    T    107;
      L     S5T#3S;
      SD    T    108;
NETWORK
TITLE =

      O     I   1042.7;
      O     I   1040.7;
      O     ;
      A     M   1030.1;
      AN    I   1040.0;
      =     M   1021.4;
NETWORK
TITLE =

      L     MD   244;
      L     L#0;
      <>D   ;
      =     M   1021.5;
NETWORK
TITLE =

      L     MD   244;
      L     L#0;
      ==D   ;
      =     M   1021.6;
NETWORK
TITLE =

      A     I   1048.0;
      L     S5T#500MS;
      SD    T    392;
      L     S5T#3S;
      SD    T    393;
NETWORK
TITLE =

      L     0;
      L     MW   184;
      <>I   ;
      =     M   1022.6;
NETWORK
TITLE =
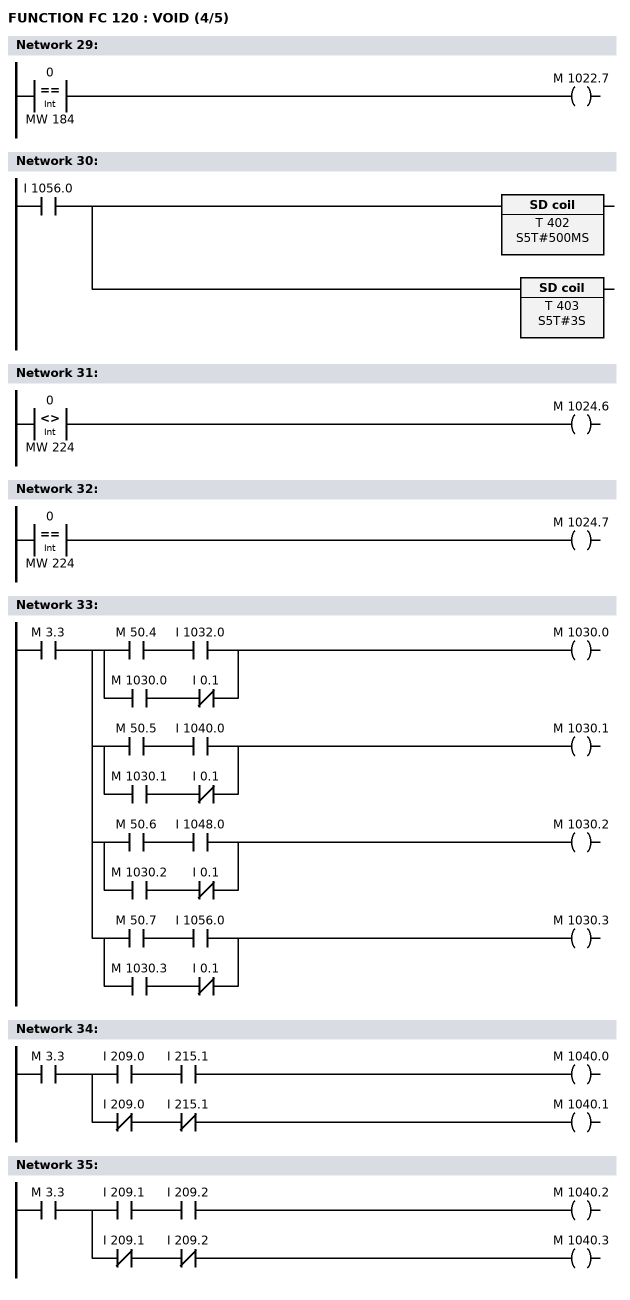

      L     0;
      L     MW   184;
      ==I   ;
      =     M   1022.7;
NETWORK
TITLE =

      A     I   1056.0;
      L     S5T#500MS;
      SD    T    402;
      L     S5T#3S;
      SD    T    403;
NETWORK
TITLE =

      L     0;
      L     MW   224;
      <>I   ;
      =     M   1024.6;
NETWORK
TITLE =

      L     0;
      L     MW   224;
      ==I   ;
      =     M   1024.7;
NETWORK
TITLE =

      A     M      3.3;
      =     L      0.0;
      A     L      0.0;
      A(    ;
      A     M     50.4;
      A     I   1032.0;
      O     ;
      A     M   1030.0;
      AN    I      0.1;
      )     ;
      =     M   1030.0;
      A     L      0.0;
      A(    ;
      A     M     50.5;
      A     I   1040.0;
      O     ;
      A     M   1030.1;
      AN    I      0.1;
      )     ;
      =     M   1030.1;
      A     L      0.0;
      A(    ;
      A     M     50.6;
      A     I   1048.0;
      O     ;
      A     M   1030.2;
      AN    I      0.1;
      )     ;
      =     M   1030.2;
      A     L      0.0;
      A(    ;
      A     M     50.7;
      A     I   1056.0;
      O     ;
      A     M   1030.3;
      AN    I      0.1;
      )     ;
      =     M   1030.3;
NETWORK
TITLE =

      A     M      3.3;
      =     L      0.0;
      A     L      0.0;
      A     I    209.0;
      A     I    215.1;
      =     M   1040.0;
      A     L      0.0;
      AN    I    209.0;
      AN    I    215.1;
      =     M   1040.1;
NETWORK
TITLE =

      A     M      3.3;
      =     L      0.0;
      A     L      0.0;
      A     I    209.1;
      A     I    209.2;
      =     M   1040.2;
      A     L      0.0;
      AN    I    209.1;
      AN    I    209.2;
      =     M   1040.3;
NETWORK
TITLE =
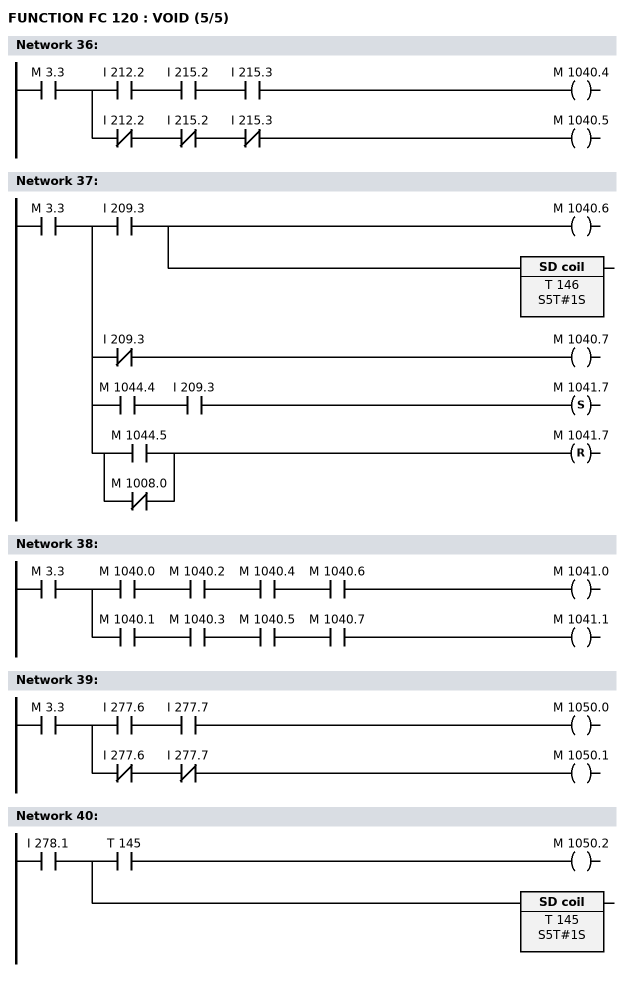

      A     M      3.3;
      =     L      0.0;
      A     L      0.0;
      A     I    212.2;
      A     I    215.2;
      A     I    215.3;
      =     M   1040.4;
      A     L      0.0;
      AN    I    212.2;
      AN    I    215.2;
      AN    I    215.3;
      =     M   1040.5;
NETWORK
TITLE =

      A     M      3.3;
      =     L      0.0;
      A     L      0.0;
      A     I    209.3;
      =     M   1040.6;
      L     S5T#1S;
      SD    T    146;
      A     L      0.0;
      AN    I    209.3;
      =     M   1040.7;
      A     L      0.0;
      A     M   1044.4;
      A     I    209.3;
      S     M   1041.7;
      A     L      0.0;
      A(    ;
      O     M   1044.5;
      ON    M   1008.0;
      )     ;
      R     M   1041.7;
NETWORK
TITLE =

      A     M      3.3;
      =     L      0.0;
      A     L      0.0;
      A     M   1040.0;
      A     M   1040.2;
      A     M   1040.4;
      A     M   1040.6;
      =     M   1041.0;
      A     L      0.0;
      A     M   1040.1;
      A     M   1040.3;
      A     M   1040.5;
      A     M   1040.7;
      =     M   1041.1;
NETWORK
TITLE =

      A     M      3.3;
      =     L      0.0;
      A     L      0.0;
      A     I    277.6;
      A     I    277.7;
      =     M   1050.0;
      A     L      0.0;
      AN    I    277.6;
      AN    I    277.7;
      =     M   1050.1;
NETWORK
TITLE =

      A     I    278.1;
      =     L      0.0;
      A     L      0.0;
      A     T    145;
      =     M   1050.2;
      A     L      0.0;
      BLD   102;
      L     S5T#1S;
      SD    T    145;
END_FUNCTION

FUNCTION_BLOCK FB 121
TITLE =
VERSION : 0.1


VAR
  S701_RETURN_LOCK_ERR : FB 424;	//S701_RETURN_LOCK_ERR
  S701_TURN_LOCK_ERR : FB 424;	//S701_TURN_LOCK_ERR
  S701_LM_PIN1_ERR : FB 424;	//S701_LM_PIN1_ERR
  S701_LM_PIN2_ERR : FB 424;	//S701_LM_PIN2_ERR
  S701_LM_PIN3_ERR : FB 424;	//S701_LM_PIN3_ERR
  S701_LM_1_CLAMP1_ERR : FB 424;	//S701_LM_1_CLAMP1_ERR
  S701_LM_1_CLAMP2_ERR : FB 424;	//S701_LM_1_CLAMP2_ERR
  S701_LM_1_CLAMP3_ERR : FB 424;	//S701_LM_1_CLAMP3_ERR
  S701_LM_1_CLAMP4_ERR : FB 424;	//S701_LM_1_CLAMP4_ERR
  S701_LM_2_CLAMP1_ERR : FB 424;	//S701_LM_2_CLAMP1_ERR
  S701_LM_2_CLAMP2_ERR : FB 424;	//S701_LM_2_CLAMP2_ERR
  S701_LM_2_CLAMP3_ERR : FB 424;	//S701_LM_2_CLAMP3_ERR
  S701_TL_PIN1_ERR : FB 424;
  S701_LM_2_CLAMP4_ERR : FB 424;	//S701_LM_2_CLAMP4_ERR
  S701_LM_2_CLAMP5_ERR : FB 424;	//S701_LM_2_CLAMP5_ERR
  S701_LM_FDR_SFT_ERR : FB 424;	//S701_LM_FDR_SFT_ERR
  S701_LM_FDR_PIN_ERR : FB 424;
  S701_TL_PIN2_ERR : FB 424;
  S701_TL_LOCATE1_ERR : FB 424;
  S701_TL_LOCATE2_ERR : FB 424;
  S701_TL_LOCATE3_ERR : FB 424;
  S701_TL_1_CLAMP1_ERR : FB 426;
  S701_TL_1_CLAMP2_ERR : FB 426;
  S701_TL_2_CLAMP_ERR : FB 426;
  S701_TL_3_CLAMP_ERR : FB 426;
  S701_TL_4_CLAMP_ERR : FB 426;
  S701_TL_FDR_SFT_ERR : FB 426;
END_VAR
BEGIN
NETWORK
TITLE =
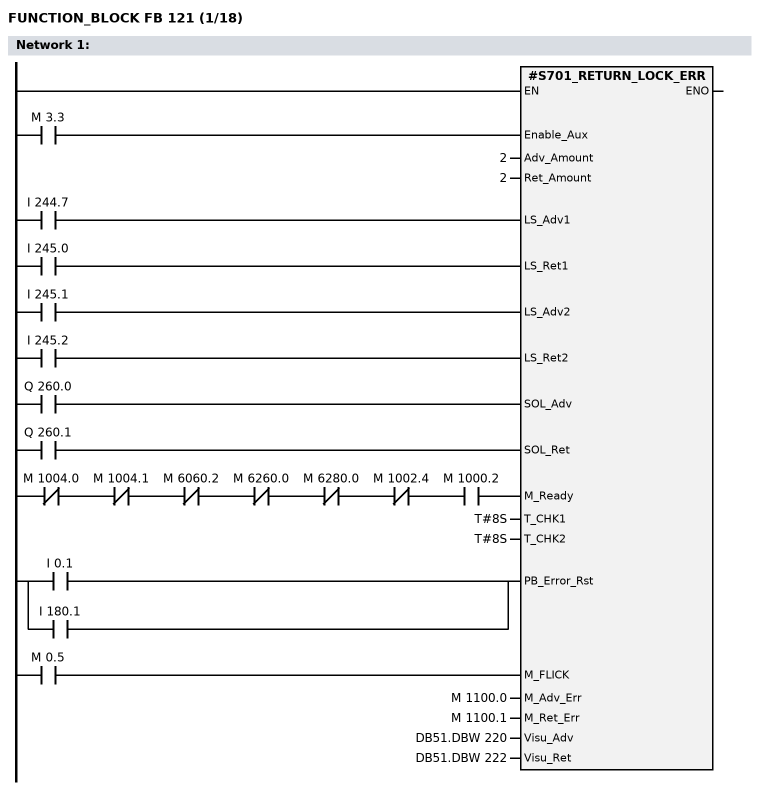

      A     M      3.3;
      =     L      0.0;
      BLD   103;
      A     I    244.7;
      =     L      0.1;
      BLD   103;
      A     I    245.0;
      =     L      0.2;
      BLD   103;
      A     I    245.1;
      =     L      0.3;
      BLD   103;
      A     I    245.2;
      =     L      0.4;
      BLD   103;
      A     Q    260.0;
      =     L      1.1;
      BLD   103;
      A     Q    260.1;
      =     L      1.2;
      BLD   103;
      AN    M   1004.0;
      AN    M   1004.1;
      AN    M   6060.2;
      AN    M   6260.0;
      AN    M   6280.0;
      AN    M   1002.4;
      A     M   1000.2;
      =     L      1.3;
      BLD   103;
      A(    ;
      O     I      0.1;
      O     I    180.1;
      )     ;
      =     L      1.5;
      BLD   103;
      A     M      0.5;
      =     L      1.6;
      BLD   103;
      CALL #S701_RETURN_LOCK_ERR (
           Enable_Aux               := L      0.0,
           Adv_Amount               := 2,
           Ret_Amount               := 2,
           LS_Adv1                  := L      0.1,
           LS_Ret1                  := L      0.2,
           LS_Adv2                  := L      0.3,
           LS_Ret2                  := L      0.4,
           SOL_Adv                  := L      1.1,
           SOL_Ret                  := L      1.2,
           M_Ready                  := L      1.3,
           T_CHK1                   := T#8S,
           T_CHK2                   := T#8S,
           PB_Error_Rst             := L      1.5,
           M_FLICK                  := L      1.6,
           M_Adv_Err                := M   1100.0,
           M_Ret_Err                := M   1100.1,
           Visu_Adv                 := DB51.DBW  220,
           Visu_Ret                 := DB51.DBW  222);
      NOP   0;
NETWORK
TITLE =
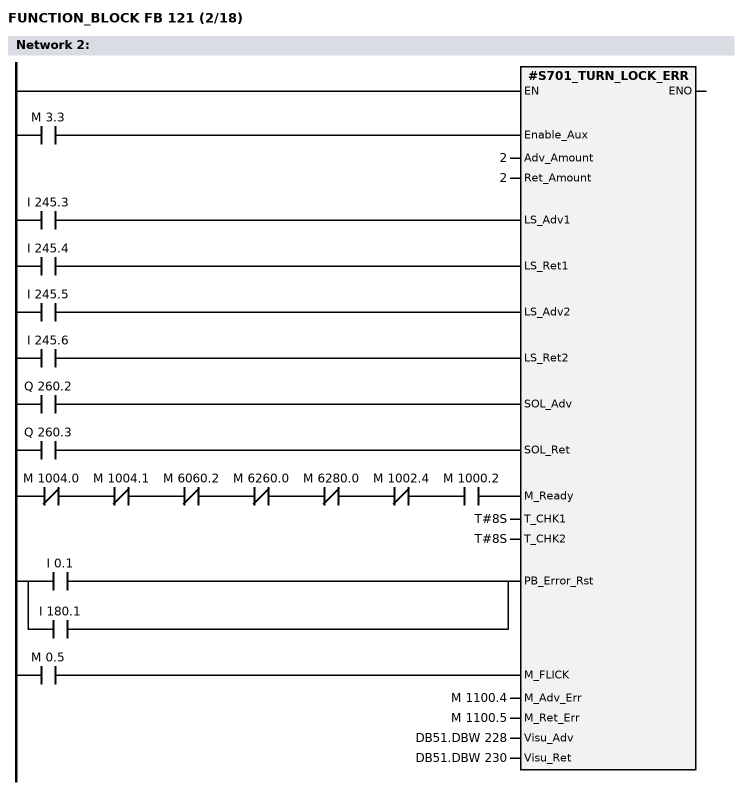

      A     M      3.3;
      =     L      0.0;
      BLD   103;
      A     I    245.3;
      =     L      0.1;
      BLD   103;
      A     I    245.4;
      =     L      0.2;
      BLD   103;
      A     I    245.5;
      =     L      0.3;
      BLD   103;
      A     I    245.6;
      =     L      0.4;
      BLD   103;
      A     Q    260.2;
      =     L      1.1;
      BLD   103;
      A     Q    260.3;
      =     L      1.2;
      BLD   103;
      AN    M   1004.0;
      AN    M   1004.1;
      AN    M   6060.2;
      AN    M   6260.0;
      AN    M   6280.0;
      AN    M   1002.4;
      A     M   1000.2;
      =     L      1.3;
      BLD   103;
      A(    ;
      O     I      0.1;
      O     I    180.1;
      )     ;
      =     L      1.5;
      BLD   103;
      A     M      0.5;
      =     L      1.6;
      BLD   103;
      CALL #S701_TURN_LOCK_ERR (
           Enable_Aux               := L      0.0,
           Adv_Amount               := 2,
           Ret_Amount               := 2,
           LS_Adv1                  := L      0.1,
           LS_Ret1                  := L      0.2,
           LS_Adv2                  := L      0.3,
           LS_Ret2                  := L      0.4,
           SOL_Adv                  := L      1.1,
           SOL_Ret                  := L      1.2,
           M_Ready                  := L      1.3,
           T_CHK1                   := T#8S,
           T_CHK2                   := T#8S,
           PB_Error_Rst             := L      1.5,
           M_FLICK                  := L      1.6,
           M_Adv_Err                := M   1100.4,
           M_Ret_Err                := M   1100.5,
           Visu_Adv                 := DB51.DBW  228,
           Visu_Ret                 := DB51.DBW  230);
      NOP   0;
NETWORK
TITLE =
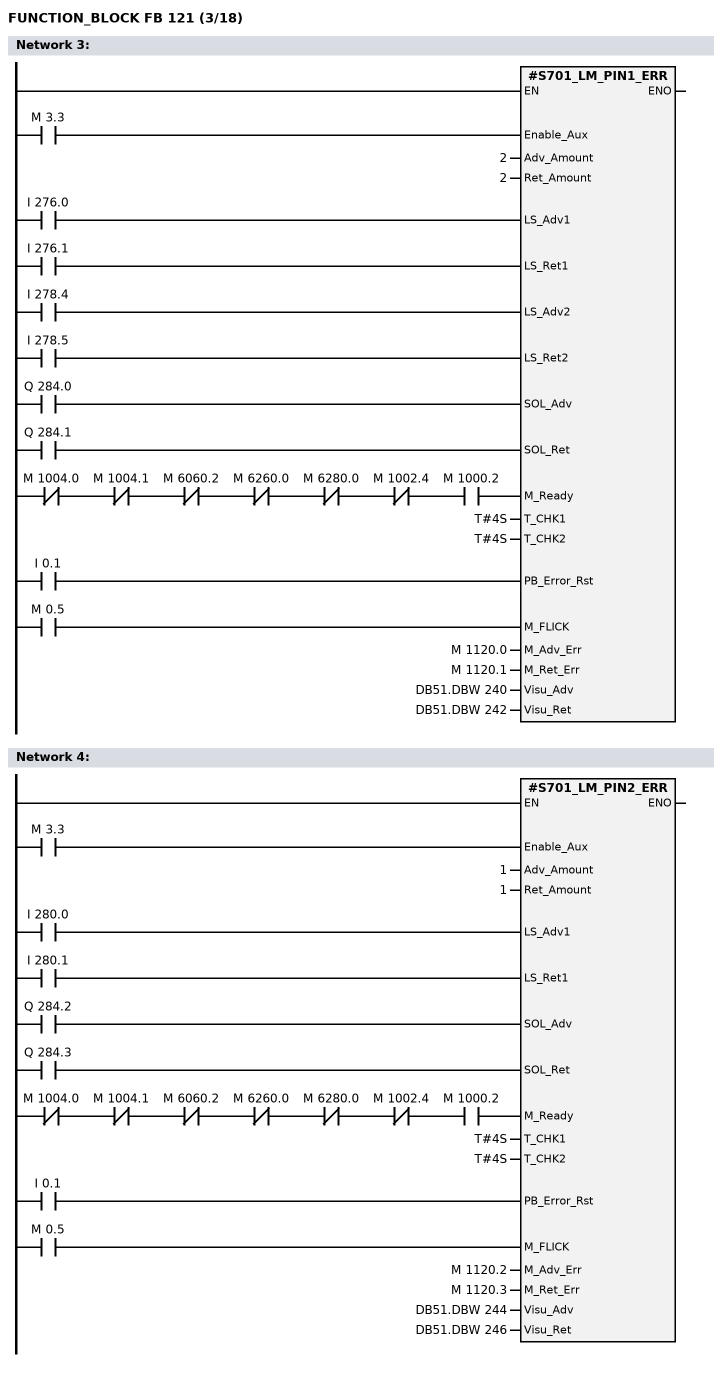

      A     M      3.3;
      =     L      0.0;
      BLD   103;
      A     I    276.0;
      =     L      0.1;
      BLD   103;
      A     I    276.1;
      =     L      0.2;
      BLD   103;
      A     I    278.4;
      =     L      0.3;
      BLD   103;
      A     I    278.5;
      =     L      0.4;
      BLD   103;
      A     Q    284.0;
      =     L      1.1;
      BLD   103;
      A     Q    284.1;
      =     L      1.2;
      BLD   103;
      AN    M   1004.0;
      AN    M   1004.1;
      AN    M   6060.2;
      AN    M   6260.0;
      AN    M   6280.0;
      AN    M   1002.4;
      A     M   1000.2;
      =     L      1.3;
      BLD   103;
      A     I      0.1;
      =     L      1.5;
      BLD   103;
      A     M      0.5;
      =     L      1.6;
      BLD   103;
      CALL #S701_LM_PIN1_ERR (
           Enable_Aux               := L      0.0,
           Adv_Amount               := 2,
           Ret_Amount               := 2,
           LS_Adv1                  := L      0.1,
           LS_Ret1                  := L      0.2,
           LS_Adv2                  := L      0.3,
           LS_Ret2                  := L      0.4,
           SOL_Adv                  := L      1.1,
           SOL_Ret                  := L      1.2,
           M_Ready                  := L      1.3,
           T_CHK1                   := T#4S,
           T_CHK2                   := T#4S,
           PB_Error_Rst             := L      1.5,
           M_FLICK                  := L      1.6,
           M_Adv_Err                := M   1120.0,
           M_Ret_Err                := M   1120.1,
           Visu_Adv                 := DB51.DBW  240,
           Visu_Ret                 := DB51.DBW  242);
      NOP   0;
NETWORK
TITLE =

      A     M      3.3;
      =     L      0.0;
      BLD   103;
      A     I    280.0;
      =     L      0.1;
      BLD   103;
      A     I    280.1;
      =     L      0.2;
      BLD   103;
      A     Q    284.2;
      =     L      1.1;
      BLD   103;
      A     Q    284.3;
      =     L      1.2;
      BLD   103;
      AN    M   1004.0;
      AN    M   1004.1;
      AN    M   6060.2;
      AN    M   6260.0;
      AN    M   6280.0;
      AN    M   1002.4;
      A     M   1000.2;
      =     L      1.3;
      BLD   103;
      A     I      0.1;
      =     L      1.5;
      BLD   103;
      A     M      0.5;
      =     L      1.6;
      BLD   103;
      CALL #S701_LM_PIN2_ERR (
           Enable_Aux               := L      0.0,
           Adv_Amount               := 1,
           Ret_Amount               := 1,
           LS_Adv1                  := L      0.1,
           LS_Ret1                  := L      0.2,
           SOL_Adv                  := L      1.1,
           SOL_Ret                  := L      1.2,
           M_Ready                  := L      1.3,
           T_CHK1                   := T#4S,
           T_CHK2                   := T#4S,
           PB_Error_Rst             := L      1.5,
           M_FLICK                  := L      1.6,
           M_Adv_Err                := M   1120.2,
           M_Ret_Err                := M   1120.3,
           Visu_Adv                 := DB51.DBW  244,
           Visu_Ret                 := DB51.DBW  246);
      NOP   0;
NETWORK
TITLE =
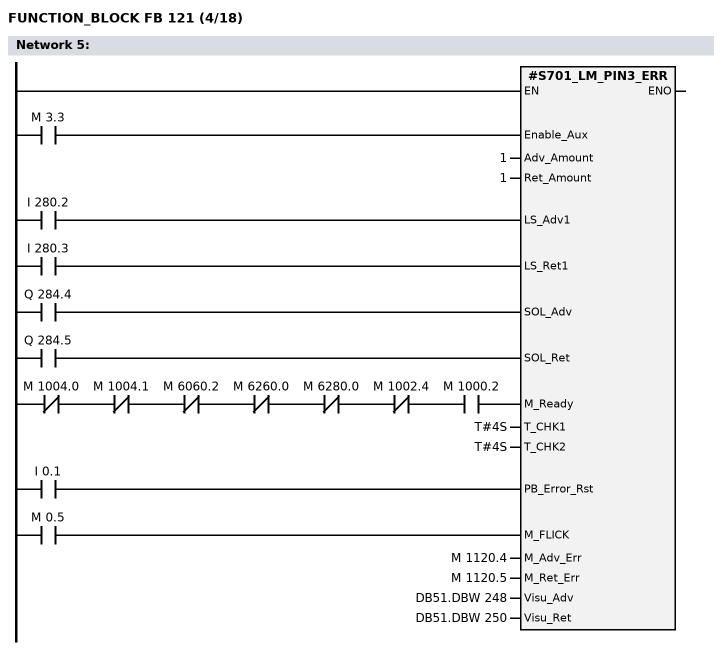

      A     M      3.3;
      =     L      0.0;
      BLD   103;
      A     I    280.2;
      =     L      0.1;
      BLD   103;
      A     I    280.3;
      =     L      0.2;
      BLD   103;
      A     Q    284.4;
      =     L      1.1;
      BLD   103;
      A     Q    284.5;
      =     L      1.2;
      BLD   103;
      AN    M   1004.0;
      AN    M   1004.1;
      AN    M   6060.2;
      AN    M   6260.0;
      AN    M   6280.0;
      AN    M   1002.4;
      A     M   1000.2;
      =     L      1.3;
      BLD   103;
      A     I      0.1;
      =     L      1.5;
      BLD   103;
      A     M      0.5;
      =     L      1.6;
      BLD   103;
      CALL #S701_LM_PIN3_ERR (
           Enable_Aux               := L      0.0,
           Adv_Amount               := 1,
           Ret_Amount               := 1,
           LS_Adv1                  := L      0.1,
           LS_Ret1                  := L      0.2,
           SOL_Adv                  := L      1.1,
           SOL_Ret                  := L      1.2,
           M_Ready                  := L      1.3,
           T_CHK1                   := T#4S,
           T_CHK2                   := T#4S,
           PB_Error_Rst             := L      1.5,
           M_FLICK                  := L      1.6,
           M_Adv_Err                := M   1120.4,
           M_Ret_Err                := M   1120.5,
           Visu_Adv                 := DB51.DBW  248,
           Visu_Ret                 := DB51.DBW  250);
      NOP   0;
NETWORK
TITLE =
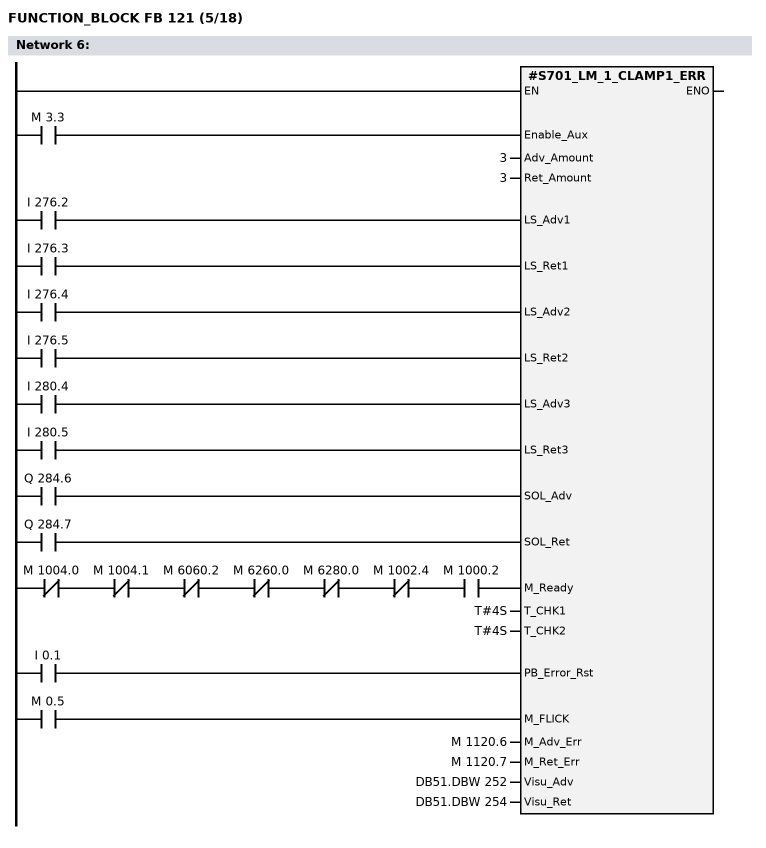

      A     M      3.3;
      =     L      0.0;
      BLD   103;
      A     I    276.2;
      =     L      0.1;
      BLD   103;
      A     I    276.3;
      =     L      0.2;
      BLD   103;
      A     I    276.4;
      =     L      0.3;
      BLD   103;
      A     I    276.5;
      =     L      0.4;
      BLD   103;
      A     I    280.4;
      =     L      0.5;
      BLD   103;
      A     I    280.5;
      =     L      0.6;
      BLD   103;
      A     Q    284.6;
      =     L      1.1;
      BLD   103;
      A     Q    284.7;
      =     L      1.2;
      BLD   103;
      AN    M   1004.0;
      AN    M   1004.1;
      AN    M   6060.2;
      AN    M   6260.0;
      AN    M   6280.0;
      AN    M   1002.4;
      A     M   1000.2;
      =     L      1.3;
      BLD   103;
      A     I      0.1;
      =     L      1.5;
      BLD   103;
      A     M      0.5;
      =     L      1.6;
      BLD   103;
      CALL #S701_LM_1_CLAMP1_ERR (
           Enable_Aux               := L      0.0,
           Adv_Amount               := 3,
           Ret_Amount               := 3,
           LS_Adv1                  := L      0.1,
           LS_Ret1                  := L      0.2,
           LS_Adv2                  := L      0.3,
           LS_Ret2                  := L      0.4,
           LS_Adv3                  := L      0.5,
           LS_Ret3                  := L      0.6,
           SOL_Adv                  := L      1.1,
           SOL_Ret                  := L      1.2,
           M_Ready                  := L      1.3,
           T_CHK1                   := T#4S,
           T_CHK2                   := T#4S,
           PB_Error_Rst             := L      1.5,
           M_FLICK                  := L      1.6,
           M_Adv_Err                := M   1120.6,
           M_Ret_Err                := M   1120.7,
           Visu_Adv                 := DB51.DBW  252,
           Visu_Ret                 := DB51.DBW  254);
      NOP   0;
NETWORK
TITLE =
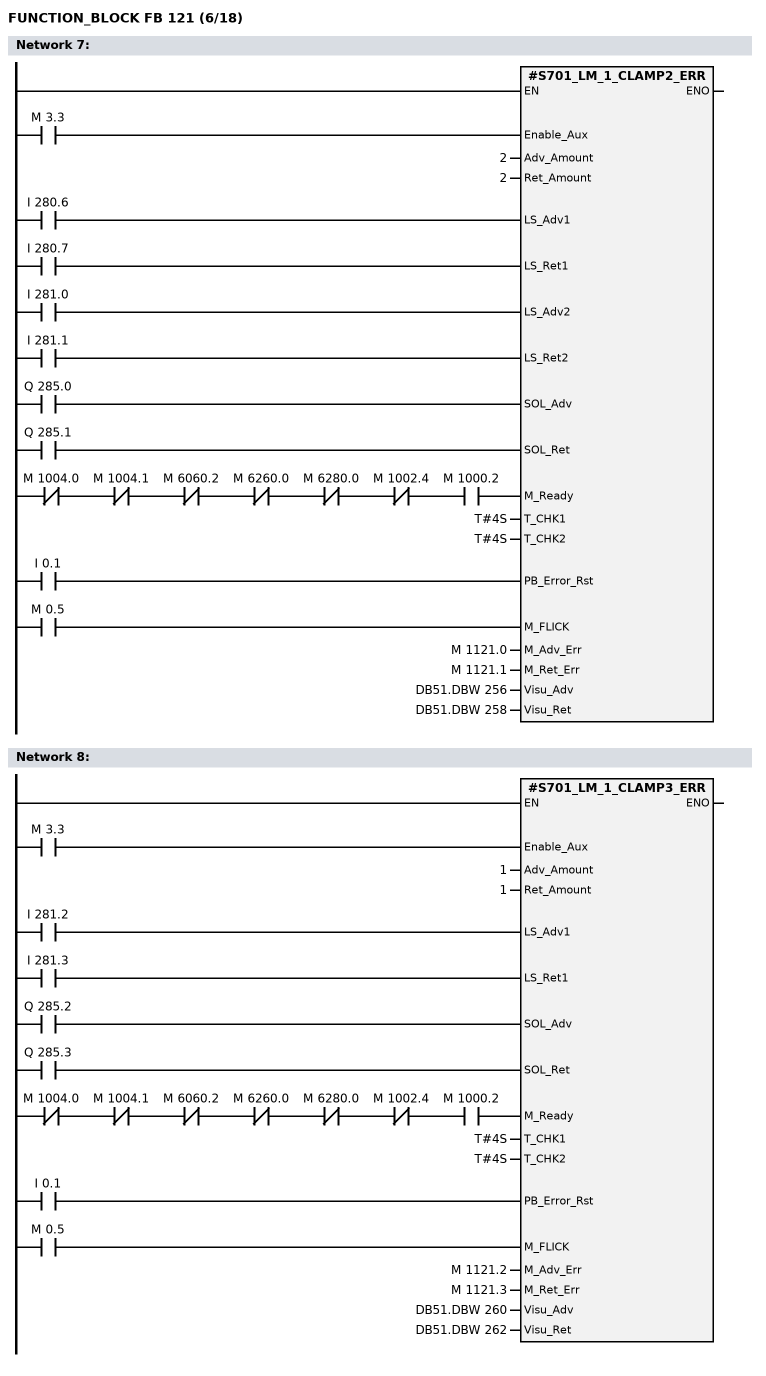

      A     M      3.3;
      =     L      0.0;
      BLD   103;
      A     I    280.6;
      =     L      0.1;
      BLD   103;
      A     I    280.7;
      =     L      0.2;
      BLD   103;
      A     I    281.0;
      =     L      0.3;
      BLD   103;
      A     I    281.1;
      =     L      0.4;
      BLD   103;
      A     Q    285.0;
      =     L      1.1;
      BLD   103;
      A     Q    285.1;
      =     L      1.2;
      BLD   103;
      AN    M   1004.0;
      AN    M   1004.1;
      AN    M   6060.2;
      AN    M   6260.0;
      AN    M   6280.0;
      AN    M   1002.4;
      A     M   1000.2;
      =     L      1.3;
      BLD   103;
      A     I      0.1;
      =     L      1.5;
      BLD   103;
      A     M      0.5;
      =     L      1.6;
      BLD   103;
      CALL #S701_LM_1_CLAMP2_ERR (
           Enable_Aux               := L      0.0,
           Adv_Amount               := 2,
           Ret_Amount               := 2,
           LS_Adv1                  := L      0.1,
           LS_Ret1                  := L      0.2,
           LS_Adv2                  := L      0.3,
           LS_Ret2                  := L      0.4,
           SOL_Adv                  := L      1.1,
           SOL_Ret                  := L      1.2,
           M_Ready                  := L      1.3,
           T_CHK1                   := T#4S,
           T_CHK2                   := T#4S,
           PB_Error_Rst             := L      1.5,
           M_FLICK                  := L      1.6,
           M_Adv_Err                := M   1121.0,
           M_Ret_Err                := M   1121.1,
           Visu_Adv                 := DB51.DBW  256,
           Visu_Ret                 := DB51.DBW  258);
      NOP   0;
NETWORK
TITLE =

      A     M      3.3;
      =     L      0.0;
      BLD   103;
      A     I    281.2;
      =     L      0.1;
      BLD   103;
      A     I    281.3;
      =     L      0.2;
      BLD   103;
      A     Q    285.2;
      =     L      1.1;
      BLD   103;
      A     Q    285.3;
      =     L      1.2;
      BLD   103;
      AN    M   1004.0;
      AN    M   1004.1;
      AN    M   6060.2;
      AN    M   6260.0;
      AN    M   6280.0;
      AN    M   1002.4;
      A     M   1000.2;
      =     L      1.3;
      BLD   103;
      A     I      0.1;
      =     L      1.5;
      BLD   103;
      A     M      0.5;
      =     L      1.6;
      BLD   103;
      CALL #S701_LM_1_CLAMP3_ERR (
           Enable_Aux               := L      0.0,
           Adv_Amount               := 1,
           Ret_Amount               := 1,
           LS_Adv1                  := L      0.1,
           LS_Ret1                  := L      0.2,
           SOL_Adv                  := L      1.1,
           SOL_Ret                  := L      1.2,
           M_Ready                  := L      1.3,
           T_CHK1                   := T#4S,
           T_CHK2                   := T#4S,
           PB_Error_Rst             := L      1.5,
           M_FLICK                  := L      1.6,
           M_Adv_Err                := M   1121.2,
           M_Ret_Err                := M   1121.3,
           Visu_Adv                 := DB51.DBW  260,
           Visu_Ret                 := DB51.DBW  262);
      NOP   0;
NETWORK
TITLE =
